LIN {X 0,Y 458.208,Z 900.819,A -85,B 0,C 180,E1 13122.077,E2 13122.077} C_VEL
LIN {X 0,Y 454.402,Z 922.56,A -85,B 0,C 180,E1 13121.642,E2 13121.642} C_VEL
LIN {X 0,Y 449.592,Z 944.659,A -85,B 0,C 180,E1 13121.087,E2 13121.087} C_VEL
LIN {X 0,Y 442.831,Z 970.318,A -85,B 0,C 180,E1 13120.289,E2 13120.289} C_VEL
LIN {X 0,Y 434.901,Z 994.961,A -85,B 0,C 180,E1 13119.322,E2 13119.322} C_VEL
LIN {X 0,Y 427.473,Z 1015.224,A -85,B 0,C 180,E1 13118.375,E2 13118.375} C_VEL
LIN {X 0,Y 419.408,Z 1034.951,A -85,B 0,C 180,E1 13117.289,E2 13117.289} C_VEL
LIN {X 0,Y 409.247,Z 1057.358,A -85,B 0,C 180,E1 13115.837,E2 13115.837} C_VEL
LIN {X 0,Y 397.642,Z 1080.077,A -85,B 0,C 180,E1 13114.053,E2 13114.053} C_VEL
LIN {X 0,Y 387.753,Z 1097.858,A -85,B 0,C 180,E1 13112.398,E2 13112.398} C_VEL
LIN {X 0,Y 377.989,Z 1114.238,A -85,B 0,C 180,E1 13110.628,E2 13110.628} C_VEL
LIN {X 0,Y 368.063,Z 1129.874,A -85,B 0,C 180,E1 13108.672,E2 13108.672} C_VEL
LIN {X 0,Y 355.822,Z 1148.166,A -85,B 0,C 180,E1 13105.975,E2 13105.975} C_VEL
LIN {X 0,Y 343.486,Z 1165.363,A -85,B 0,C 180,E1 13102.886,E2 13102.886} C_VEL
LIN {X 0,Y 333.685,Z 1178.527,A -85,B 0,C 180,E1 13100.078,E2 13100.078} C_VEL
LIN {X 0,Y 324.574,Z 1190.478,A -85,B 0,C 180,E1 13097.092,E2 13097.092} C_VEL
LIN {X 0,Y 315.879,Z 1201.713,A -85,B 0,C 180,E1 13093.803,E2 13093.803} C_VEL
LIN {X 0,Y 306.032,Z 1214.541,A -85,B 0,C 180,E1 13089.321,E2 13089.321} C_VEL
LIN {X 0,Y 297.777,Z 1225.367,A -85,B 0,C 180,E1 13084.561,E2 13084.561} C_VEL
LIN {X 0,Y 292.177,Z 1233.181,A -85,B 0,C 180,E1 13080.413,E2 13080.413} C_VEL
LIN {X 0,Y 287.782,Z 1239.822,A -85,B 0,C 180,E1 13076.172,E2 13076.172} C_VEL
LIN {X 0,Y 284.237,Z 1245.857,A -85,B 0,C 180,E1 13071.449,E2 13071.449} C_VEL
LIN {X 0,Y 281.638,Z 1251.335,A -85,B 0,C 180,E1 13065.819,E2 13065.819} C_VEL
LIN {X 0,Y 280.53,Z 1254.566,A -85,B 0,C 180,E1 13061.087,E2 13061.087} C_VEL
LIN {X 0,Y 280.133,Z 1256.541,A -85,B 0,C 180,E1 13056.755,E2 13056.755} C_VEL
LIN {X 0,Y 280.008,Z 1257.539,A -85,B 0,C 180,E1 13052.651,E2 13052.651} C_VEL
LIN {X 0,Y 279.986,Z 1257.679,A -85,B 0,C 180,E1 13048.558,E2 13048.558} C_VEL
LIN {X 0,Y 280.068,Z 1256.959,A -85,B 0,C 180,E1 13044.459,E2 13044.459} C_VEL
LIN {X 0,Y 280.331,Z 1255.374,A -85,B 0,C 180,E1 13040.34,E2 13040.34} C_VEL
LIN {X 0,Y 281.103,Z 1252.753,A -85,B 0,C 180,E1 13035.994,E2 13035.994} C_VEL
LIN {X 0,Y 282.595,Z 1249.134,A -85,B 0,C 180,E1 13031.636,E2 13031.636} C_VEL
LIN {X 0,Y 284.991,Z 1244.486,A -85,B 0,C 180,E1 13027.29,E2 13027.29} C_VEL
LIN {X 0,Y 288.66,Z 1238.479,A -85,B 0,C 180,E1 13022.783,E2 13022.783} C_VEL
LIN {X 0,Y 294.638,Z 1229.864,A -85,B 0,C 180,E1 13017.567,E2 13017.567} C_VEL
LIN {X 0,Y 302.104,Z 1219.641,A -85,B 0,C 180,E1 13012.714,E2 13012.714} C_VEL
LIN {X 0,Y 309.339,Z 1210.213,A -85,B 0,C 180,E1 13008.984,E2 13008.984} C_VEL
LIN {X 0,Y 317.621,Z 1199.529,A -85,B 0,C 180,E1 13005.403,E2 13005.403} C_VEL
LIN {X 0,Y 328.464,Z 1185.62,A -85,B 0,C 180,E1 13001.5,E2 13001.5} C_VEL
LIN {X 0,Y 340.404,Z 1169.657,A -85,B 0,C 180,E1 12997.873,E2 12997.873} C_VEL
LIN {X 0,Y 350.282,Z 1156.036,A -85,B 0,C 180,E1 12995.266,E2 12995.266} C_VEL
LIN {X 0,Y 359.989,Z 1142.109,A -85,B 0,C 180,E1 12992.976,E2 12992.976} C_VEL
LIN {X 0,Y 370.544,Z 1126.229,A -85,B 0,C 180,E1 12990.737,E2 12990.737} C_VEL
LIN {X 0,Y 383.441,Z 1105.562,A -85,B 0,C 180,E1 12988.284,E2 12988.284} C_VEL
LIN {X 0,Y 394.996,Z 1085.203,A -85,B 0,C 180,E1 12986.295,E2 12986.295} C_VEL
LIN {X 0,Y 404.338,Z 1067.469,A -85,B 0,C 180,E1 12984.822,E2 12984.822} C_VEL
LIN {X 0,Y 412.871,Z 1049.87,A -85,B 0,C 180,E1 12983.553,E2 12983.553} C_VEL
LIN {X 0,Y 416.305,Z 1042.588,A -85,B 0,C 180,E1 12983.075,E2 12983.075} C_VEL
LIN {X 0,Y 418.753,Z 1036.276,A -85,B 0,C 180,E1 12982.553,E2 12982.553} C_VEL
LIN {X 0,Y 423.276,Z 1019.851,A -85,B 0,C 180,E1 12980.83,E2 12980.83} C_VEL
LIN {X 0,Y 425.239,Z 1014.185,A -85,B 0,C 180,E1 12980.445,E2 12980.445} C_VEL
LIN {X 0,Y 433.639,Z 991.447,A -85,B 0,C 180,E1 12979.417,E2 12979.417} C_VEL
LIN {X 0,Y 441.922,Z 964.972,A -85,B 0,C 180,E1 12978.443,E2 12978.443} C_VEL
LIN {X 0,Y 447.766,Z 942.648,A -85,B 0,C 180,E1 12977.78,E2 12977.78} C_VEL
LIN {X 0,Y 452.432,Z 921.238,A -85,B 0,C 180,E1 12977.26,E2 12977.26} C_VEL
LIN {X 0,Y 456.431,Z 898.287,A -85,B 0,C 180,E1 12976.818,E2 12976.818} C_VEL
LIN {X 0,Y 460.408,Z 864.162,A -85,B 0,C 180,E1 12976.277,E2 12976.277} C_VEL
LIN {X 0,Y 479.796,Z 660.807,A -85,B 0,C 180,E1 12973.266,E2 12973.266} C_VEL
LIN {X 0,Y 476.185,Z 654.134,A -85,B 0,C 180,E1 12970.71,E2 12970.71} C_VEL
LIN {X 0,Y 473.814,Z 649.968,A -85,B 0,C 180,E1 12968.617,E2 12968.617} C_VEL
LIN {X 0,Y 471.686,Z 646,A -85,B 0,C 180,E1 12966.084,E2 12966.084} C_VEL
LIN {X 0,Y 469.89,Z 641.972,A -85,B 0,C 180,E1 12961.829,E2 12961.829} C_VEL
LIN {X 0,Y 469.82,Z 641.352,A -85,B 0,C 180,E1 12960.976,E2 12960.976} C_VEL
LIN {X 0,Y 469.873,Z 641.573,A -85,B 0,C 180,E1 12958.903,E2 12958.903} C_VEL
LIN {X 0,Y 471.37,Z 645.689,A -85,B 0,C 180,E1 12954.767,E2 12954.767} C_VEL
LIN {X 0,Y 472.117,Z 646.8,A -85,B 0,C 180,E1 12953.738,E2 12953.738} C_VEL
LIN {X 0,Y 474.753,Z 651.624,A -85,B 0,C 180,E1 12950.912,E2 12950.912} C_VEL
LIN {X 0,Y 477.243,Z 656.203,A -85,B 0,C 180,E1 12948.886,E2 12948.886} C_VEL
LIN {X 0,Y 479.059,Z 659.618,A -85,B 0,C 180,E1 12947.616,E2 12947.616} C_VEL
LIN {X 0,Y 479.91,Z 661.708,A -85,B 0,C 180,E1 12947.034,E2 12947.034} C_VEL
LIN {X 0,Y 459.294,Z 878.88,A -85,B 0,C 180,E1 12943.812,E2 12943.812} C_VEL
LIN {X 0,Y 455.731,Z 908,A -85,B 0,C 180,E1 12943.338,E2 12943.338} C_VEL
LIN {X 0,Y 451.723,Z 930.654,A -85,B 0,C 180,E1 12942.918,E2 12942.918} C_VEL
LIN {X 0,Y 446.837,Z 952.503,A -85,B 0,C 180,E1 12942.435,E2 12942.435} C_VEL
LIN {X 0,Y 440.026,Z 977.894,A -85,B 0,C 180,E1 12941.725,E2 12941.725} C_VEL
LIN {X 0,Y 431.647,Z 1003.54,A -85,B 0,C 180,E1 12940.813,E2 12940.813} C_VEL
LIN {X 0,Y 423.793,Z 1024.563,A -85,B 0,C 180,E1 12939.899,E2 12939.899} C_VEL
LIN {X 0,Y 415.815,Z 1043.731,A -85,B 0,C 180,E1 12938.917,E2 12938.917} C_VEL
LIN {X 0,Y 406.864,Z 1063.298,A -85,B 0,C 180,E1 12937.736,E2 12937.736} C_VEL
LIN {X 0,Y 395.004,Z 1086.874,A -85,B 0,C 180,E1 12936.046,E2 12936.046} C_VEL
LIN {X 0,Y 382.76,Z 1108.625,A -85,B 0,C 180,E1 12934.135,E2 12934.135} C_VEL
LIN {X 0,Y 372.487,Z 1125.659,A -85,B 0,C 180,E1 12932.364,E2 12932.364} C_VEL
LIN {X 0,Y 361.948,Z 1142.122,A -85,B 0,C 180,E1 12930.364,E2 12930.364} C_VEL
LIN {X 0,Y 349.824,Z 1160.077,A -85,B 0,C 180,E1 12927.793,E2 12927.793} C_VEL
LIN {X 0,Y 336.403,Z 1178.724,A -85,B 0,C 180,E1 12924.538,E2 12924.538} C_VEL
LIN {X 0,Y 326.264,Z 1192.331,A -85,B 0,C 180,E1 12921.688,E2 12921.688} C_VEL
LIN {X 0,Y 316.923,Z 1204.607,A -85,B 0,C 180,E1 12918.676,E2 12918.676} C_VEL
LIN {X 0,Y 307.429,Z 1216.966,A -85,B 0,C 180,E1 12915.107,E2 12915.107} C_VEL
LIN {X 0,Y 296.996,Z 1230.755,A -85,B 0,C 180,E1 12910.279,E2 12910.279} C_VEL
LIN {X 0,Y 289.063,Z 1241.475,A -85,B 0,C 180,E1 12905.621,E2 12905.621} C_VEL
LIN {X 0,Y 283.333,Z 1249.819,A -85,B 0,C 180,E1 12901.258,E2 12901.258} C_VEL
LIN {X 0,Y 278.777,Z 1257.144,A -85,B 0,C 180,E1 12896.646,E2 12896.646} C_VEL
LIN {X 0,Y 274.966,Z 1264.468,A -85,B 0,C 180,E1 12890.886,E2 12890.886} C_VEL
LIN {X 0,Y 273.019,Z 1269.339,A -85,B 0,C 180,E1 12885.734,E2 12885.734} C_VEL
LIN {X 0,Y 272.243,Z 1272.504,A -85,B 0,C 180,E1 12881.234,E2 12881.234} C_VEL
LIN {X 0,Y 272.013,Z 1274.548,A -85,B 0,C 180,E1 12876.977,E2 12876.977} C_VEL
LIN {X 0,Y 271.992,Z 1275.618,A -85,B 0,C 180,E1 12872.96,E2 12872.96} C_VEL
LIN {X 0,Y 271.98,Z 1275.809,A -85,B 0,C 180,E1 12868.746,E2 12868.746} C_VEL
LIN {X 0,Y 271.99,Z 1275.049,A -85,B 0,C 180,E1 12864.525,E2 12864.525} C_VEL
LIN {X 0,Y 272.086,Z 1273.337,A -85,B 0,C 180,E1 12860.278,E2 12860.278} C_VEL
LIN {X 0,Y 272.693,Z 1270.509,A -85,B 0,C 180,E1 12855.789,E2 12855.789} C_VEL
LIN {X 0,Y 274.01,Z 1266.621,A -85,B 0,C 180,E1 12851.28,E2 12851.28} C_VEL
LIN {X 0,Y 276.262,Z 1261.652,A -85,B 0,C 180,E1 12846.776,E2 12846.776} C_VEL
LIN {X 0,Y 279.474,Z 1255.891,A -85,B 0,C 180,E1 12842.526,E2 12842.526} C_VEL
LIN {X 0,Y 284.029,Z 1248.723,A -85,B 0,C 180,E1 12838.139,E2 12838.139} C_VEL
LIN {X 0,Y 291.432,Z 1238.275,A -85,B 0,C 180,E1 12832.868,E2 12832.868} C_VEL
LIN {X 0,Y 300.371,Z 1226.138,A -85,B 0,C 180,E1 12828.017,E2 12828.017} C_VEL
LIN {X 0,Y 308.826,Z 1215.076,A -85,B 0,C 180,E1 12824.329,E2 12824.329} C_VEL
LIN {X 0,Y 318.374,Z 1202.649,A -85,B 0,C 180,E1 12820.826,E2 12820.826} C_VEL
LIN {X 0,Y 330.9,Z 1186.15,A -85,B 0,C 180,E1 12816.965,E2 12816.965} C_VEL
LIN {X 0,Y 342.902,Z 1169.616,A -85,B 0,C 180,E1 12813.812,E2 12813.812} C_VEL
LIN {X 0,Y 353.575,Z 1154.399,A -85,B 0,C 180,E1 12811.366,E2 12811.366} C_VEL
LIN {X 0,Y 364.164,Z 1138.584,A -85,B 0,C 180,E1 12809.196,E2 12809.196} C_VEL
LIN {X 0,Y 377.019,Z 1118.286,A -85,B 0,C 180,E1 12806.842,E2 12806.842} C_VEL
LIN {X 0,Y 389.335,Z 1096.889,A -85,B 0,C 180,E1 12804.812,E2 12804.812} C_VEL
LIN {X 0,Y 399.1,Z 1078.591,A -85,B 0,C 180,E1 12803.34,E2 12803.34} C_VEL
LIN {X 0,Y 408.668,Z 1059.163,A -85,B 0,C 180,E1 12802.008,E2 12802.008} C_VEL
LIN {X 0,Y 418.509,Z 1037.249,A -85,B 0,C 180,E1 12800.74,E2 12800.74} C_VEL
LIN {X 0,Y 428.549,Z 1011.748,A -85,B 0,C 180,E1 12799.533,E2 12799.533} C_VEL
LIN {X 0,Y 435.907,Z 990.374,A -85,B 0,C 180,E1 12798.705,E2 12798.705} C_VEL
LIN {X 0,Y 441.98,Z 970.274,A -85,B 0,C 180,E1 12798.055,E2 12798.055} C_VEL
LIN {X 0,Y 447.636,Z 948.487,A -85,B 0,C 180,E1 12797.476,E2 12797.476} C_VEL
LIN {X 0,Y 453.046,Z 923.261,A -85,B 0,C 180,E1 12796.943,E2 12796.943} C_VEL
LIN {X 0,Y 457.356,Z 894.787,A -85,B 0,C 180,E1 12796.445,E2 12796.445} C_VEL
LIN {X 0,Y 464.969,Z 816.08,A -85,B 0,C 180,E1 12795.257,E2 12795.257} C_VEL
LIN {X 0,Y 479.707,Z 661.387,A -85,B 0,C 180,E1 12792.948,E2 12792.948} C_VEL
LIN {X 0,Y 477.878,Z 657.566,A -85,B 0,C 180,E1 12791.71,E2 12791.71} C_VEL
LIN {X 0,Y 475.155,Z 652.651,A -85,B 0,C 180,E1 12789.631,E2 12789.631} C_VEL
LIN {X 0,Y 473.644,Z 649.962,A -85,B 0,C 180,E1 12788.253,E2 12788.253} C_VEL
LIN {X 0,Y 471.486,Z 645.953,A -85,B 0,C 180,E1 12785.72,E2 12785.72} C_VEL
LIN {X 0,Y 469.719,Z 642.322,A -85,B 0,C 180,E1 12781.952,E2 12781.952} C_VEL
LIN {X 0,Y 469.602,Z 641.325,A -85,B 0,C 180,E1 12780.976,E2 12780.976} C_VEL
LIN {X 0,Y 469.642,Z 641.564,A -85,B 0,C 180,E1 12778.17,E2 12778.17} C_VEL
LIN {X 0,Y 471.383,Z 645.828,A -85,B 0,C 180,E1 12773.912,E2 12773.912} C_VEL
LIN {X 0,Y 472.055,Z 647.057,A -85,B 0,C 180,E1 12773.004,E2 12773.004} C_VEL
LIN {X 0,Y 474.46,Z 651.334,A -85,B 0,C 180,E1 12770.478,E2 12770.478} C_VEL
LIN {X 0,Y 477.27,Z 656.469,A -85,B 0,C 180,E1 12768.213,E2 12768.213} C_VEL
LIN {X 0,Y 479.605,Z 660.806,A -85,B 0,C 180,E1 12766.635,E2 12766.635} C_VEL
LIN {X 0,Y 458.7,Z 879.164,A -85,B 0,C 180,E1 12763.397,E2 12763.397} C_VEL
LIN {X 0,Y 455.655,Z 902.058,A -85,B 0,C 180,E1 12763.018,E2 12763.018} C_VEL
LIN {X 0,Y 451.751,Z 923.802,A -85,B 0,C 180,E1 12762.585,E2 12762.585} C_VEL
LIN {X 0,Y 446.411,Z 947.667,A -85,B 0,C 180,E1 12761.986,E2 12761.986} C_VEL
LIN {X 0,Y 438.836,Z 974.812,A -85,B 0,C 180,E1 12761.122,E2 12761.122} C_VEL
LIN {X 0,Y 431.717,Z 996.356,A -85,B 0,C 180,E1 12760.275,E2 12760.275} C_VEL
LIN {X 0,Y 424.163,Z 1016.494,A -85,B 0,C 180,E1 12759.34,E2 12759.34} C_VEL
LIN {X 0,Y 416.019,Z 1035.968,A -85,B 0,C 180,E1 12758.276,E2 12758.276} C_VEL
LIN {X 0,Y 404.868,Z 1059.921,A -85,B 0,C 180,E1 12756.725,E2 12756.725} C_VEL
LIN {X 0,Y 393.273,Z 1081.892,A -85,B 0,C 180,E1 12754.989,E2 12754.989} C_VEL
LIN {X 0,Y 383.503,Z 1099.004,A -85,B 0,C 180,E1 12753.395,E2 12753.395} C_VEL
LIN {X 0,Y 373.675,Z 1115.061,A -85,B 0,C 180,E1 12751.663,E2 12751.663} C_VEL
LIN {X 0,Y 362.847,Z 1131.649,A -85,B 0,C 180,E1 12749.581,E2 12749.581} C_VEL
LIN {X 0,Y 349.383,Z 1151.011,A -85,B 0,C 180,E1 12746.667,E2 12746.667} C_VEL
LIN {X 0,Y 337.953,Z 1166.396,A -85,B 0,C 180,E1 12743.855,E2 12743.855} C_VEL
LIN {X 0,Y 327.862,Z 1179.49,A -85,B 0,C 180,E1 12741.032,E2 12741.032} C_VEL
LIN {X 0,Y 318.054,Z 1191.887,A -85,B 0,C 180,E1 12737.88,E2 12737.88} C_VEL
LIN {X 0,Y 307.077,Z 1205.615,A -85,B 0,C 180,E1 12733.708,E2 12733.708} C_VEL
LIN {X 0,Y 297.378,Z 1217.505,A -85,B 0,C 180,E1 12729.193,E2 12729.193} C_VEL
LIN {X 0,Y 290.336,Z 1226.43,A -85,B 0,C 180,E1 12725.095,E2 12725.095} C_VEL
LIN {X 0,Y 284.549,Z 1234.133,A -85,B 0,C 180,E1 12720.853,E2 12720.853} C_VEL
LIN {X 0,Y 279.442,Z 1241.562,A -85,B 0,C 180,E1 12715.871,E2 12715.871} C_VEL
LIN {X 0,Y 275.381,Z 1248.326,A -85,B 0,C 180,E1 12709.945,E2 12709.945} C_VEL
LIN {X 0,Y 273.434,Z 1252.438,A -85,B 0,C 180,E1 12705.117,E2 12705.117} C_VEL
LIN {X 0,Y 272.515,Z 1255.049,A -85,B 0,C 180,E1 12700.989,E2 12700.989} C_VEL
LIN {X 0,Y 272.138,Z 1256.869,A -85,B 0,C 180,E1 12696.742,E2 12696.742} C_VEL
LIN {X 0,Y 272.013,Z 1257.802,A -85,B 0,C 180,E1 12692.729,E2 12692.729} C_VEL
LIN {X 0,Y 271.983,Z 1257.964,A -85,B 0,C 180,E1 12688.727,E2 12688.727} C_VEL
LIN {X 0,Y 272.072,Z 1257.287,A -85,B 0,C 180,E1 12684.508,E2 12684.508} C_VEL
LIN {X 0,Y 272.363,Z 1255.639,A -85,B 0,C 180,E1 12680.055,E2 12680.055} C_VEL
LIN {X 0,Y 273.215,Z 1253.019,A -85,B 0,C 180,E1 12675.581,E2 12675.581} C_VEL
LIN {X 0,Y 274.835,Z 1249.378,A -85,B 0,C 180,E1 12671.071,E2 12671.071} C_VEL
LIN {X 0,Y 277.395,Z 1244.756,A -85,B 0,C 180,E1 12666.632,E2 12666.632} C_VEL
LIN {X 0,Y 281.107,Z 1239.043,A -85,B 0,C 180,E1 12662.219,E2 12662.219} C_VEL
LIN {X 0,Y 287.107,Z 1230.825,A -85,B 0,C 180,E1 12657.069,E2 12657.069} C_VEL
LIN {X 0,Y 295.163,Z 1220.361,A -85,B 0,C 180,E1 12651.927,E2 12651.927} C_VEL
LIN {X 0,Y 303.082,Z 1210.485,A -85,B 0,C 180,E1 12647.947,E2 12647.947} C_VEL
LIN {X 0,Y 311.727,Z 1199.801,A -85,B 0,C 180,E1 12644.325,E2 12644.325} C_VEL
LIN {X 0,Y 323.002,Z 1185.891,A -85,B 0,C 180,E1 12640.393,E2 12640.393} C_VEL
LIN {X 0,Y 334.962,Z 1170.462,A -85,B 0,C 180,E1 12636.861,E2 12636.861} C_VEL
LIN {X 0,Y 345.562,Z 1156.305,A -85,B 0,C 180,E1 12634.144,E2 12634.144} C_VEL
LIN {X 0,Y 356.201,Z 1141.464,A -85,B 0,C 180,E1 12631.72,E2 12631.72} C_VEL
LIN {X 0,Y 368.389,Z 1123.555,A -85,B 0,C 180,E1 12629.246,E2 12629.246} C_VEL
LIN {X 0,Y 381.61,Z 1102.427,A -85,B 0,C 180,E1 12626.844,E2 12626.844} C_VEL
LIN {X 0,Y 392.067,Z 1084.328,A -85,B 0,C 180,E1 12625.12,E2 12625.12} C_VEL
LIN {X 0,Y 401.727,Z 1066.276,A -85,B 0,C 180,E1 12623.651,E2 12623.651} C_VEL
LIN {X 0,Y 410.852,Z 1047.707,A -85,B 0,C 180,E1 12622.352,E2 12622.352} C_VEL
LIN {X 0,Y 421.721,Z 1023.115,A -85,B 0,C 180,E1 12620.898,E2 12620.898} C_VEL
LIN {X 0,Y 425.239,Z 1014.185,A -85,B 0,C 180,E1 12620.445,E2 12620.445} C_VEL
LIN {X 0,Y 427.575,Z 1007.549,A -85,B 0,C 180,E1 12619.999,E2 12619.999} C_VEL
LIN {X 0,Y 431.528,Z 991.264,A -85,B 0,C 180,E1 12618.513,E2 12618.513} C_VEL
LIN {X 0,Y 433.488,Z 984.381,A -85,B 0,C 180,E1 12618.119,E2 12618.119} C_VEL
LIN {X 0,Y 440.062,Z 963.018,A -85,B 0,C 180,E1 12617.378,E2 12617.378} C_VEL
LIN {X 0,Y 445.664,Z 941.713,A -85,B 0,C 180,E1 12616.764,E2 12616.764} C_VEL
LIN {X 0,Y 450.436,Z 919.913,A -85,B 0,C 180,E1 12616.252,E2 12616.252} C_VEL
LIN {X 0,Y 455.094,Z 892.816,A -85,B 0,C 180,E1 12615.752,E2 12615.752} C_VEL
LIN {X 0,Y 459.703,Z 848.917,A -85,B 0,C 180,E1 12615.086,E2 12615.086} C_VEL
LIN {X 0,Y 477.447,Z 666.619,A -85,B 0,C 180,E1 12612.402,E2 12612.402} C_VEL
LIN {X 0,Y 474.383,Z 661,A -85,B 0,C 180,E1 12610.076,E2 12610.076} C_VEL
LIN {X 0,Y 472.589,Z 657.681,A -85,B 0,C 180,E1 12608.395,E2 12608.395} C_VEL
LIN {X 0,Y 470.622,Z 653.883,A -85,B 0,C 180,E1 12605.976,E2 12605.976} C_VEL
LIN {X 0,Y 468.896,Z 649.851,A -85,B 0,C 180,E1 12601.711,E2 12601.711} C_VEL
LIN {X 0,Y 468.833,Z 649.296,A -85,B 0,C 180,E1 12600.855,E2 12600.855} C_VEL
LIN {X 0,Y 468.888,Z 649.598,A -85,B 0,C 180,E1 12598.9,E2 12598.9} C_VEL
LIN {X 0,Y 470.395,Z 653.667,A -85,B 0,C 180,E1 12594.756,E2 12594.756} C_VEL
LIN {X 0,Y 471.081,Z 654.828,A -85,B 0,C 180,E1 12593.786,E2 12593.786} C_VEL
LIN {X 0,Y 473.565,Z 659.444,A -85,B 0,C 180,E1 12591.072,E2 12591.072} C_VEL
LIN {X 0,Y 476.005,Z 664.046,A -85,B 0,C 180,E1 12589.041,E2 12589.041} C_VEL
LIN {X 0,Y 477.6,Z 667.148,A -85,B 0,C 180,E1 12587.894,E2 12587.894} C_VEL
LIN {X 0,Y 456.821,Z 881.666,A -85,B 0,C 180,E1 12584.736,E2 12584.736} C_VEL
LIN {X 0,Y 453.331,Z 908.729,A -85,B 0,C 180,E1 12584.296,E2 12584.296} C_VEL
LIN {X 0,Y 449.294,Z 931.036,A -85,B 0,C 180,E1 12583.887,E2 12583.887} C_VEL
LIN {X 0,Y 444.21,Z 953.307,A -85,B 0,C 180,E1 12583.401,E2 12583.401} C_VEL
LIN {X 0,Y 436.833,Z 980.014,A -85,B 0,C 180,E1 12582.658,E2 12582.658} C_VEL
LIN {X 0,Y 428.5,Z 1004.768,A -85,B 0,C 180,E1 12581.779,E2 12581.779} C_VEL
LIN {X 0,Y 421.059,Z 1024.302,A -85,B 0,C 180,E1 12580.941,E2 12580.941} C_VEL
LIN {X 0,Y 412.941,Z 1043.468,A -85,B 0,C 180,E1 12579.977,E2 12579.977} C_VEL
LIN {X 0,Y 403.697,Z 1063.286,A -85,B 0,C 180,E1 12578.8,E2 12578.8} C_VEL
LIN {X 0,Y 391.722,Z 1086.607,A -85,B 0,C 180,E1 12577.151,E2 12577.151} C_VEL
LIN {X 0,Y 379.266,Z 1108.269,A -85,B 0,C 180,E1 12575.271,E2 12575.271} C_VEL
LIN {X 0,Y 368.342,Z 1125.951,A -85,B 0,C 180,E1 12573.447,E2 12573.447} C_VEL
LIN {X 0,Y 357.473,Z 1142.472,A -85,B 0,C 180,E1 12571.446,E2 12571.446} C_VEL
LIN {X 0,Y 344.129,Z 1161.658,A -85,B 0,C 180,E1 12568.684,E2 12568.684} C_VEL
LIN {X 0,Y 330.986,Z 1179.233,A -85,B 0,C 180,E1 12565.569,E2 12565.569} C_VEL
LIN {X 0,Y 320.542,Z 1192.769,A -85,B 0,C 180,E1 12562.706,E2 12562.706} C_VEL
LIN {X 0,Y 310.381,Z 1205.626,A -85,B 0,C 180,E1 12559.497,E2 12559.497} C_VEL
LIN {X 0,Y 298.908,Z 1220.065,A -85,B 0,C 180,E1 12555.176,E2 12555.176} C_VEL
LIN {X 0,Y 288.683,Z 1232.832,A -85,B 0,C 180,E1 12550.377,E2 12550.377} C_VEL
LIN {X 0,Y 281.829,Z 1241.758,A -85,B 0,C 180,E1 12546.343,E2 12546.343} C_VEL
LIN {X 0,Y 275.935,Z 1249.908,A -85,B 0,C 180,E1 12541.95,E2 12541.95} C_VEL
LIN {X 0,Y 270.788,Z 1257.81,A -85,B 0,C 180,E1 12536.784,E2 12536.784} C_VEL
LIN {X 0,Y 266.909,Z 1264.843,A -85,B 0,C 180,E1 12530.857,E2 12530.857} C_VEL
LIN {X 0,Y 265.074,Z 1269.238,A -85,B 0,C 180,E1 12525.993,E2 12525.993} C_VEL
LIN {X 0,Y 264.272,Z 1272.283,A -85,B 0,C 180,E1 12521.493,E2 12521.493} C_VEL
LIN {X 0,Y 264.019,Z 1274.301,A -85,B 0,C 180,E1 12517.138,E2 12517.138} C_VEL
LIN {X 0,Y 263.995,Z 1275.355,A -85,B 0,C 180,E1 12513.049,E2 12513.049} C_VEL
LIN {X 0,Y 263.986,Z 1275.546,A -85,B 0,C 180,E1 12508.708,E2 12508.708} C_VEL
LIN {X 0,Y 263.994,Z 1274.785,A -85,B 0,C 180,E1 12504.359,E2 12504.359} C_VEL
LIN {X 0,Y 264.107,Z 1273.071,A -85,B 0,C 180,E1 12499.981,E2 12499.981} C_VEL
LIN {X 0,Y 264.777,Z 1270.24,A -85,B 0,C 180,E1 12495.355,E2 12495.355} C_VEL
LIN {X 0,Y 266.215,Z 1266.349,A -85,B 0,C 180,E1 12490.711,E2 12490.711} C_VEL
LIN {X 0,Y 268.649,Z 1261.379,A -85,B 0,C 180,E1 12486.078,E2 12486.078} C_VEL
LIN {X 0,Y 272.078,Z 1255.615,A -85,B 0,C 180,E1 12481.714,E2 12481.714} C_VEL
LIN {X 0,Y 276.916,Z 1248.445,A -85,B 0,C 180,E1 12477.219,E2 12477.219} C_VEL
LIN {X 0,Y 284.745,Z 1237.996,A -85,B 0,C 180,E1 12471.842,E2 12471.842} C_VEL
LIN {X 0,Y 294.143,Z 1225.859,A -85,B 0,C 180,E1 12466.916,E2 12466.916} C_VEL
LIN {X 0,Y 302.986,Z 1214.797,A -85,B 0,C 180,E1 12463.186,E2 12463.186} C_VEL
LIN {X 0,Y 312.522,Z 1202.855,A -85,B 0,C 180,E1 12459.783,E2 12459.783} C_VEL
LIN {X 0,Y 325.254,Z 1186.74,A -85,B 0,C 180,E1 12455.957,E2 12455.957} C_VEL
LIN {X 0,Y 337.665,Z 1170.196,A -85,B 0,C 180,E1 12452.776,E2 12452.776} C_VEL
LIN {X 0,Y 348.727,Z 1154.907,A -85,B 0,C 180,E1 12450.307,E2 12450.307} C_VEL
LIN {X 0,Y 359.467,Z 1139.333,A -85,B 0,C 180,E1 12448.166,E2 12448.166} C_VEL
LIN {X 0,Y 370.356,Z 1122.62,A -85,B 0,C 180,E1 12446.202,E2 12446.202} C_VEL
LIN {X 0,Y 384.054,Z 1099.985,A -85,B 0,C 180,E1 12443.984,E2 12443.984} C_VEL
LIN {X 0,Y 395.093,Z 1079.872,A -85,B 0,C 180,E1 12442.358,E2 12442.358} C_VEL
LIN {X 0,Y 404.869,Z 1060.524,A -85,B 0,C 180,E1 12441.035,E2 12441.035} C_VEL
LIN {X 0,Y 414.021,Z 1040.69,A -85,B 0,C 180,E1 12439.884,E2 12439.884} C_VEL
LIN {X 0,Y 424.257,Z 1016.016,A -85,B 0,C 180,E1 12438.689,E2 12438.689} C_VEL
LIN {X 0,Y 432.956,Z 991.392,A -85,B 0,C 180,E1 12437.733,E2 12437.733} C_VEL
LIN {X 0,Y 439.337,Z 970.713,A -85,B 0,C 180,E1 12437.073,E2 12437.073} C_VEL
LIN {X 0,Y 444.987,Z 949.409,A -85,B 0,C 180,E1 12436.514,E2 12436.514} C_VEL
LIN {X 0,Y 449.988,Z 926.777,A -85,B 0,C 180,E1 12436.037,E2 12436.037} C_VEL
LIN {X 0,Y 454.779,Z 897.617,A -85,B 0,C 180,E1 12435.522,E2 12435.522} C_VEL
LIN {X 0,Y 459.902,Z 847.321,A -85,B 0,C 180,E1 12434.762,E2 12434.762} C_VEL
LIN {X 0,Y 477.403,Z 667.033,A -85,B 0,C 180,E1 12432.107,E2 12432.107} C_VEL
LIN {X 0,Y 474.528,Z 661.442,A -85,B 0,C 180,E1 12429.95,E2 12429.95} C_VEL
LIN {X 0,Y 472.415,Z 657.674,A -85,B 0,C 180,E1 12428.03,E2 12428.03} C_VEL
LIN {X 0,Y 470.42,Z 653.834,A -85,B 0,C 180,E1 12425.611,E2 12425.611} C_VEL
LIN {X 0,Y 468.698,Z 650.05,A -85,B 0,C 180,E1 12421.711,E2 12421.711} C_VEL
LIN {X 0,Y 468.606,Z 649.27,A -85,B 0,C 180,E1 12420.856,E2 12420.856} C_VEL
LIN {X 0,Y 468.648,Z 649.446,A -85,B 0,C 180,E1 12418.288,E2 12418.288} C_VEL
LIN {X 0,Y 470.32,Z 653.709,A -85,B 0,C 180,E1 12414.02,E2 12414.02} C_VEL
LIN {X 0,Y 471.11,Z 655.294,A -85,B 0,C 180,E1 12412.929,E2 12412.929} C_VEL
LIN {X 0,Y 473.272,Z 659.16,A -85,B 0,C 180,E1 12410.637,E2 12410.637} C_VEL
LIN {X 0,Y 475.949,Z 664.164,A -85,B 0,C 180,E1 12408.426,E2 12408.426} C_VEL
LIN {X 0,Y 477.259,Z 666.712,A -85,B 0,C 180,E1 12407.488,E2 12407.488} C_VEL
LIN {X 0,Y 456.221,Z 881.637,A -85,B 0,C 180,E1 12404.326,E2 12404.326} C_VEL
LIN {X 0,Y 453.147,Z 903.794,A -85,B 0,C 180,E1 12403.96,E2 12403.96} C_VEL
LIN {X 0,Y 448.892,Z 926.703,A -85,B 0,C 180,E1 12403.502,E2 12403.502} C_VEL
LIN {X 0,Y 442.081,Z 955.209,A -85,B 0,C 180,E1 12402.765,E2 12402.765} C_VEL
LIN {X 0,Y 435.6,Z 977.25,A -85,B 0,C 180,E1 12402.044,E2 12402.044} C_VEL
LIN {X 0,Y 428.653,Z 997.752,A -85,B 0,C 180,E1 12401.242,E2 12401.242} C_VEL
LIN {X 0,Y 420.899,Z 1017.956,A -85,B 0,C 180,E1 12400.311,E2 12400.311} C_VEL
LIN {X 0,Y 411.308,Z 1040.285,A -85,B 0,C 180,E1 12399.084,E2 12399.084} C_VEL
LIN {X 0,Y 399.507,Z 1064.363,A -85,B 0,C 180,E1 12397.485,E2 12397.485} C_VEL
LIN {X 0,Y 389.136,Z 1083.487,A -85,B 0,C 180,E1 12395.964,E2 12395.964} C_VEL
LIN {X 0,Y 378.843,Z 1101.022,A -85,B 0,C 180,E1 12394.328,E2 12394.328} C_VEL
LIN {X 0,Y 367.209,Z 1119.444,A -85,B 0,C 180,E1 12392.309,E2 12392.309} C_VEL
LIN {X 0,Y 353.371,Z 1139.589,A -85,B 0,C 180,E1 12389.637,E2 12389.637} C_VEL
LIN {X 0,Y 342.352,Z 1154.615,A -85,B 0,C 180,E1 12387.242,E2 12387.242} C_VEL
LIN {X 0,Y 331.925,Z 1168.187,A -85,B 0,C 180,E1 12384.704,E2 12384.704} C_VEL
LIN {X 0,Y 321.58,Z 1181.142,A -85,B 0,C 180,E1 12381.856,E2 12381.856} C_VEL
LIN {X 0,Y 310.005,Z 1195.277,A -85,B 0,C 180,E1 12378.148,E2 12378.148} C_VEL
LIN {X 0,Y 298.311,Z 1209.064,A -85,B 0,C 180,E1 12373.653,E2 12373.653} C_VEL
LIN {X 0,Y 290.028,Z 1218.88,A -85,B 0,C 180,E1 12369.753,E2 12369.753} C_VEL
LIN {X 0,Y 282.826,Z 1227.611,A -85,B 0,C 180,E1 12365.597,E2 12365.597} C_VEL
LIN {X 0,Y 276.179,Z 1236.122,A -85,B 0,C 180,E1 12360.683,E2 12360.683} C_VEL
LIN {X 0,Y 270.548,Z 1243.945,A -85,B 0,C 180,E1 12354.906,E2 12354.906} C_VEL
LIN {X 0,Y 267.329,Z 1249.192,A -85,B 0,C 180,E1 12349.888,E2 12349.888} C_VEL
LIN {X 0,Y 265.481,Z 1252.915,A -85,B 0,C 180,E1 12345.275,E2 12345.275} C_VEL
LIN {X 0,Y 264.54,Z 1255.423,A -85,B 0,C 180,E1 12341.104,E2 12341.104} C_VEL
LIN {X 0,Y 264.143,Z 1257.198,A -85,B 0,C 180,E1 12336.729,E2 12336.729} C_VEL
LIN {X 0,Y 264.016,Z 1258.086,A -85,B 0,C 180,E1 12332.595,E2 12332.595} C_VEL
LIN {X 0,Y 263.997,Z 1258.204,A -85,B 0,C 180,E1 12328.471,E2 12328.471} C_VEL
LIN {X 0,Y 264.084,Z 1257.55,A -85,B 0,C 180,E1 12324.341,E2 12324.341} C_VEL
LIN {X 0,Y 264.4,Z 1255.904,A -85,B 0,C 180,E1 12319.752,E2 12319.752} C_VEL
LIN {X 0,Y 265.338,Z 1253.286,A -85,B 0,C 180,E1 12315.143,E2 12315.143} C_VEL
LIN {X 0,Y 267.074,Z 1249.671,A -85,B 0,C 180,E1 12310.527,E2 12310.527} C_VEL
LIN {X 0,Y 269.834,Z 1245.027,A -85,B 0,C 180,E1 12305.936,E2 12305.936} C_VEL
LIN {X 0,Y 273.794,Z 1239.314,A -85,B 0,C 180,E1 12301.409,E2 12301.409} C_VEL
LIN {X 0,Y 280.129,Z 1231.119,A -85,B 0,C 180,E1 12296.154,E2 12296.154} C_VEL
LIN {X 0,Y 288.692,Z 1220.574,A -85,B 0,C 180,E1 12290.881,E2 12290.881} C_VEL
LIN {X 0,Y 296.924,Z 1210.758,A -85,B 0,C 180,E1 12286.865,E2 12286.865} C_VEL
LIN {X 0,Y 305.953,Z 1200.073,A -85,B 0,C 180,E1 12283.206,E2 12283.206} C_VEL
LIN {X 0,Y 317.666,Z 1186.161,A -85,B 0,C 180,E1 12279.248,E2 12279.248} C_VEL
LIN {X 0,Y 330.043,Z 1170.732,A -85,B 0,C 180,E1 12275.707,E2 12275.707} C_VEL
LIN {X 0,Y 340.979,Z 1156.575,A -85,B 0,C 180,E1 12272.991,E2 12272.991} C_VEL
LIN {X 0,Y 351.986,Z 1141.65,A -85,B 0,C 180,E1 12270.563,E2 12270.563} C_VEL
LIN {X 0,Y 364.478,Z 1123.761,A -85,B 0,C 180,E1 12268.108,E2 12268.108} C_VEL
LIN {X 0,Y 377.613,Z 1103.294,A -85,B 0,C 180,E1 12265.795,E2 12265.795} C_VEL
LIN {X 0,Y 388.29,Z 1085.253,A -85,B 0,C 180,E1 12264.085,E2 12264.085} C_VEL
LIN {X 0,Y 398.139,Z 1067.267,A -85,B 0,C 180,E1 12262.631,E2 12262.631} C_VEL
LIN {X 0,Y 407.044,Z 1049.578,A -85,B 0,C 180,E1 12261.4,E2 12261.4} C_VEL
LIN {X 0,Y 416.5,Z 1028.913,A -85,B 0,C 180,E1 12260.161,E2 12260.161} C_VEL
LIN {X 0,Y 426.951,Z 1002.939,A -85,B 0,C 180,E1 12258.881,E2 12258.881} C_VEL
LIN {X 0,Y 433.488,Z 984.381,A -85,B 0,C 180,E1 12258.119,E2 12258.119} C_VEL
LIN {X 0,Y 435.46,Z 977.419,A -85,B 0,C 180,E1 12257.744,E2 12257.744} C_VEL
LIN {X 0,Y 439.077,Z 959.392,A -85,B 0,C 180,E1 12256.354,E2 12256.354} C_VEL
LIN {X 0,Y 440.585,Z 953.296,A -85,B 0,C 180,E1 12256.074,E2 12256.074} C_VEL
LIN {X 0,Y 447.07,Z 925.986,A -85,B 0,C 180,E1 12255.392,E2 12255.392} C_VEL
LIN {X 0,Y 451.261,Z 903.636,A -85,B 0,C 180,E1 12254.957,E2 12254.957} C_VEL
LIN {X 0,Y 454.386,Z 881.336,A -85,B 0,C 180,E1 12254.596,E2 12254.596} C_VEL
LIN {X 0,Y 475.219,Z 672.666,A -85,B 0,C 180,E1 12251.553,E2 12251.553} C_VEL
LIN {X 0,Y 472.842,Z 668.2,A -85,B 0,C 180,E1 12249.617,E2 12249.617} C_VEL
LIN {X 0,Y 471.371,Z 665.393,A -85,B 0,C 180,E1 12248.171,E2 12248.171} C_VEL
LIN {X 0,Y 469.56,Z 661.765,A -85,B 0,C 180,E1 12245.867,E2 12245.867} C_VEL
LIN {X 0,Y 467.903,Z 657.731,A -85,B 0,C 180,E1 12241.592,E2 12241.592} C_VEL
LIN {X 0,Y 467.858,Z 657.236,A -85,B 0,C 180,E1 12240.857,E2 12240.857} C_VEL
LIN {X 0,Y 467.899,Z 657.478,A -85,B 0,C 180,E1 12239.02,E2 12239.02} C_VEL
LIN {X 0,Y 469.337,Z 661.547,A -85,B 0,C 180,E1 12234.866,E2 12234.866} C_VEL
LIN {X 0,Y 470.004,Z 662.741,A -85,B 0,C 180,E1 12233.894,E2 12233.894} C_VEL
LIN {X 0,Y 472.318,Z 667.131,A -85,B 0,C 180,E1 12231.294,E2 12231.294} C_VEL
LIN {X 0,Y 474.849,Z 672.034,A -85,B 0,C 180,E1 12229.137,E2 12229.137} C_VEL
LIN {X 0,Y 475.349,Z 673.141,A -85,B 0,C 180,E1 12228.751,E2 12228.751} C_VEL
LIN {X 0,Y 454.141,Z 886.693,A -85,B 0,C 180,E1 12225.633,E2 12225.633} C_VEL
LIN {X 0,Y 450.979,Z 909.945,A -85,B 0,C 180,E1 12225.255,E2 12225.255} C_VEL
LIN {X 0,Y 446.844,Z 932.147,A -85,B 0,C 180,E1 12224.852,E2 12224.852} C_VEL
LIN {X 0,Y 441.082,Z 956.667,A -85,B 0,C 180,E1 12224.317,E2 12224.317} C_VEL
LIN {X 0,Y 433.124,Z 983.859,A -85,B 0,C 180,E1 12223.545,E2 12223.545} C_VEL
LIN {X 0,Y 425.739,Z 1005.288,A -85,B 0,C 180,E1 12222.787,E2 12222.787} C_VEL
LIN {X 0,Y 418.051,Z 1025.051,A -85,B 0,C 180,E1 12221.95,E2 12221.95} C_VEL
LIN {X 0,Y 409.393,Z 1045.018,A -85,B 0,C 180,E1 12220.953,E2 12220.953} C_VEL
LIN {X 0,Y 398.414,Z 1067.916,A -85,B 0,C 180,E1 12219.583,E2 12219.583} C_VEL
LIN {X 0,Y 385.855,Z 1091.057,A -85,B 0,C 180,E1 12217.892,E2 12217.892} C_VEL
LIN {X 0,Y 375.114,Z 1109.23,A -85,B 0,C 180,E1 12216.303,E2 12216.303} C_VEL
LIN {X 0,Y 364.332,Z 1126.243,A -85,B 0,C 180,E1 12214.555,E2 12214.555} C_VEL
LIN {X 0,Y 352.851,Z 1143.227,A -85,B 0,C 180,E1 12212.503,E2 12212.503} C_VEL
LIN {X 0,Y 337.842,Z 1163.96,A -85,B 0,C 180,E1 12209.467,E2 12209.467} C_VEL
LIN {X 0,Y 325.909,Z 1179.456,A -85,B 0,C 180,E1 12206.69,E2 12206.69} C_VEL
LIN {X 0,Y 315.214,Z 1192.852,A -85,B 0,C 180,E1 12203.842,E2 12203.842} C_VEL
LIN {X 0,Y 304.432,Z 1205.998,A -85,B 0,C 180,E1 12200.529,E2 12200.529} C_VEL
LIN {X 0,Y 292.079,Z 1220.847,A -85,B 0,C 180,E1 12195.974,E2 12195.974} C_VEL
LIN {X 0,Y 282.309,Z 1232.556,A -85,B 0,C 180,E1 12191.486,E2 12191.486} C_VEL
LIN {X 0,Y 275.084,Z 1241.482,A -85,B 0,C 180,E1 12187.384,E2 12187.384} C_VEL
LIN {X 0,Y 268.835,Z 1249.633,A -85,B 0,C 180,E1 12182.899,E2 12182.899} C_VEL
LIN {X 0,Y 263.543,Z 1257.224,A -85,B 0,C 180,E1 12177.827,E2 12177.827} C_VEL
LIN {X 0,Y 259.195,Z 1264.572,A -85,B 0,C 180,E1 12171.508,E2 12171.508} C_VEL
LIN {X 0,Y 257.201,Z 1268.969,A -85,B 0,C 180,E1 12166.496,E2 12166.496} C_VEL
LIN {X 0,Y 256.317,Z 1271.971,A -85,B 0,C 180,E1 12161.942,E2 12161.942} C_VEL
LIN {X 0,Y 256.017,Z 1274.019,A -85,B 0,C 180,E1 12157.415,E2 12157.415} C_VEL
LIN {X 0,Y 255.998,Z 1275.092,A -85,B 0,C 180,E1 12153.145,E2 12153.145} C_VEL
LIN {X 0,Y 255.983,Z 1275.307,A -85,B 0,C 180,E1 12148.891,E2 12148.891} C_VEL
LIN {X 0,Y 255.997,Z 1274.593,A -85,B 0,C 180,E1 12144.407,E2 12144.407} C_VEL
LIN {X 0,Y 256.135,Z 1272.801,A -85,B 0,C 180,E1 12139.658,E2 12139.658} C_VEL
LIN {X 0,Y 256.864,Z 1269.962,A -85,B 0,C 180,E1 12134.882,E2 12134.882} C_VEL
LIN {X 0,Y 258.45,Z 1266.046,A -85,B 0,C 180,E1 12130.072,E2 12130.072} C_VEL
LIN {X 0,Y 261.077,Z 1261.106,A -85,B 0,C 180,E1 12125.339,E2 12125.339} C_VEL
LIN {X 0,Y 264.913,Z 1255.091,A -85,B 0,C 180,E1 12120.679,E2 12120.679} C_VEL
LIN {X 0,Y 270.441,Z 1247.44,A -85,B 0,C 180,E1 12115.821,E2 12115.821} C_VEL
LIN {X 0,Y 279.605,Z 1235.815,A -85,B 0,C 180,E1 12109.932,E2 12109.932} C_VEL
LIN {X 0,Y 288.466,Z 1225.053,A -85,B 0,C 180,E1 12105.575,E2 12105.575} C_VEL
LIN {X 0,Y 297.266,Z 1214.518,A -85,B 0,C 180,E1 12101.998,E2 12101.998} C_VEL
LIN {X 0,Y 307.587,Z 1202.09,A -85,B 0,C 180,E1 12098.442,E2 12098.442} C_VEL
LIN {X 0,Y 321.185,Z 1185.383,A -85,B 0,C 180,E1 12094.513,E2 12094.513} C_VEL
LIN {X 0,Y 333.838,Z 1169.049,A -85,B 0,C 180,E1 12091.41,E2 12091.41} C_VEL
LIN {X 0,Y 345.137,Z 1153.843,A -85,B 0,C 180,E1 12088.987,E2 12088.987} C_VEL
LIN {X 0,Y 356.661,Z 1137.515,A -85,B 0,C 180,E1 12086.782,E2 12086.782} C_VEL
LIN {X 0,Y 370.577,Z 1116.453,A -85,B 0,C 180,E1 12084.412,E2 12084.412} C_VEL
LIN {X 0,Y 383.064,Z 1095.663,A -85,B 0,C 180,E1 12082.504,E2 12082.504} C_VEL
LIN {X 0,Y 392.957,Z 1077.869,A -85,B 0,C 180,E1 12081.121,E2 12081.121} C_VEL
LIN {X 0,Y 402.8,Z 1058.614,A -85,B 0,C 180,E1 12079.841,E2 12079.841} C_VEL
LIN {X 0,Y 413.001,Z 1036.702,A -85,B 0,C 180,E1 12078.618,E2 12078.618} C_VEL
LIN {X 0,Y 423.43,Z 1011.077,A -85,B 0,C 180,E1 12077.452,E2 12077.452} C_VEL
LIN {X 0,Y 430.977,Z 989.825,A -85,B 0,C 180,E1 12076.661,E2 12076.661} C_VEL
LIN {X 0,Y 437.245,Z 969.691,A -85,B 0,C 180,E1 12076.038,E2 12076.038} C_VEL
LIN {X 0,Y 442.951,Z 948.372,A -85,B 0,C 180,E1 12075.495,E2 12075.495} C_VEL
LIN {X 0,Y 448.253,Z 924.46,A -85,B 0,C 180,E1 12075.008,E2 12075.008} C_VEL
LIN {X 0,Y 452.982,Z 894.861,A -85,B 0,C 180,E1 12074.501,E2 12074.501} C_VEL
LIN {X 0,Y 459.867,Z 826.99,A -85,B 0,C 180,E1 12073.492,E2 12073.492} C_VEL
LIN {X 0,Y 475.139,Z 672.818,A -85,B 0,C 180,E1 12071.231,E2 12071.231} C_VEL
LIN {X 0,Y 472.36,Z 667.508,A -85,B 0,C 180,E1 12068.951,E2 12068.951} C_VEL
LIN {X 0,Y 471.075,Z 665.204,A -85,B 0,C 180,E1 12067.685,E2 12067.685} C_VEL
LIN {X 0,Y 469.355,Z 661.715,A -85,B 0,C 180,E1 12065.501,E2 12065.501} C_VEL
LIN {X 0,Y 467.698,Z 657.93,A -85,B 0,C 180,E1 12061.593,E2 12061.593} C_VEL
LIN {X 0,Y 467.612,Z 657.216,A -85,B 0,C 180,E1 12060.735,E2 12060.735} C_VEL
LIN {X 0,Y 467.656,Z 657.329,A -85,B 0,C 180,E1 12058.407,E2 12058.407} C_VEL
LIN {X 0,Y 469.346,Z 661.686,A -85,B 0,C 180,E1 12054.008,E2 12054.008} C_VEL
LIN {X 0,Y 472.028,Z 666.85,A -85,B 0,C 180,E1 12050.859,E2 12050.859} C_VEL
LIN {X 0,Y 474.713,Z 672.006,A -85,B 0,C 180,E1 12048.58,E2 12048.58} C_VEL
LIN {X 0,Y 475.001,Z 672.79,A -85,B 0,C 180,E1 12048.347,E2 12048.347} C_VEL
LIN {X 0,Y 453.907,Z 883.737,A -85,B 0,C 180,E1 12045.27,E2 12045.27} C_VEL
LIN {X 0,Y 450.578,Z 906.663,A -85,B 0,C 180,E1 12044.893,E2 12044.893} C_VEL
LIN {X 0,Y 445.048,Z 934.578,A -85,B 0,C 180,E1 12044.315,E2 12044.315} C_VEL
LIN {X 0,Y 438.841,Z 958.715,A -85,B 0,C 180,E1 12043.668,E2 12043.668} C_VEL
LIN {X 0,Y 432.768,Z 978.8,A -85,B 0,C 180,E1 12043.012,E2 12043.012} C_VEL
LIN {X 0,Y 426.127,Z 998.024,A -85,B 0,C 180,E1 12042.269,E2 12042.269} C_VEL
LIN {X 0,Y 418.321,Z 1018.036,A -85,B 0,C 180,E1 12041.364,E2 12041.364} C_VEL
LIN {X 0,Y 408.624,Z 1040.231,A -85,B 0,C 180,E1 12040.168,E2 12040.168} C_VEL
LIN {X 0,Y 396.677,Z 1064.225,A -85,B 0,C 180,E1 12038.604,E2 12038.604} C_VEL
LIN {X 0,Y 386.263,Z 1083.098,A -85,B 0,C 180,E1 12037.128,E2 12037.128} C_VEL
LIN {X 0,Y 376.074,Z 1100.152,A -85,B 0,C 180,E1 12035.568,E2 12035.568} C_VEL
LIN {X 0,Y 365.427,Z 1116.705,A -85,B 0,C 180,E1 12033.806,E2 12033.806} C_VEL
LIN {X 0,Y 352.017,Z 1136.195,A -85,B 0,C 180,E1 12031.344,E2 12031.344} C_VEL
LIN {X 0,Y 338.589,Z 1154.058,A -85,B 0,C 180,E1 12028.568,E2 12028.568} C_VEL
LIN {X 0,Y 327.803,Z 1167.705,A -85,B 0,C 180,E1 12026.046,E2 12026.046} C_VEL
LIN {X 0,Y 316.971,Z 1180.856,A -85,B 0,C 180,E1 12023.176,E2 12023.176} C_VEL
LIN {X 0,Y 306.059,Z 1193.685,A -85,B 0,C 180,E1 12019.843,E2 12019.843} C_VEL
LIN {X 0,Y 293.007,Z 1208.597,A -85,B 0,C 180,E1 12015.058,E2 12015.058} C_VEL
LIN {X 0,Y 283.834,Z 1218.951,A -85,B 0,C 180,E1 12010.923,E2 12010.923} C_VEL
LIN {X 0,Y 276.54,Z 1227.373,A -85,B 0,C 180,E1 12006.871,E2 12006.871} C_VEL
LIN {X 0,Y 269.874,Z 1235.367,A -85,B 0,C 180,E1 12002.23,E2 12002.23} C_VEL
LIN {X 0,Y 263.469,Z 1243.726,A -85,B 0,C 180,E1 11996.106,E2 11996.106} C_VEL
LIN {X 0,Y 259.723,Z 1249.3,A -85,B 0,C 180,E1 11990.688,E2 11990.688} C_VEL
LIN {X 0,Y 257.688,Z 1253.031,A -85,B 0,C 180,E1 11985.98,E2 11985.98} C_VEL
LIN {X 0,Y 256.609,Z 1255.689,A -85,B 0,C 180,E1 11981.451,E2 11981.451} C_VEL
LIN {X 0,Y 256.171,Z 1257.398,A -85,B 0,C 180,E1 11977.164,E2 11977.164} C_VEL
LIN {X 0,Y 256.025,Z 1258.328,A -85,B 0,C 180,E1 11972.9,E2 11972.9} C_VEL
LIN {X 0,Y 255.995,Z 1258.488,A -85,B 0,C 180,E1 11968.647,E2 11968.647} C_VEL
LIN {X 0,Y 256.098,Z 1257.814,A -85,B 0,C 180,E1 11964.164,E2 11964.164} C_VEL
LIN {X 0,Y 256.418,Z 1256.278,A -85,B 0,C 180,E1 11959.657,E2 11959.657} C_VEL
LIN {X 0,Y 257.407,Z 1253.706,A -85,B 0,C 180,E1 11954.905,E2 11954.905} C_VEL
LIN {X 0,Y 259.239,Z 1250.138,A -85,B 0,C 180,E1 11950.149,E2 11950.149} C_VEL
LIN {X 0,Y 262.149,Z 1245.542,A -85,B 0,C 180,E1 11945.424,E2 11945.424} C_VEL
LIN {X 0,Y 266.085,Z 1240.172,A -85,B 0,C 180,E1 11940.994,E2 11940.994} C_VEL
LIN {X 0,Y 271.729,Z 1233.144,A -85,B 0,C 180,E1 11936.266,E2 11936.266} C_VEL
LIN {X 0,Y 280.341,Z 1223.144,A -85,B 0,C 180,E1 11930.844,E2 11930.844} C_VEL
LIN {X 0,Y 290.082,Z 1211.949,A -85,B 0,C 180,E1 11926.088,E2 11926.088} C_VEL
LIN {X 0,Y 299.308,Z 1201.468,A -85,B 0,C 180,E1 11922.405,E2 11922.405} C_VEL
LIN {X 0,Y 309.147,Z 1190.171,A -85,B 0,C 180,E1 11919.073,E2 11919.073} C_VEL
LIN {X 0,Y 321.658,Z 1175.47,A -85,B 0,C 180,E1 11915.459,E2 11915.459} C_VEL
LIN {X 0,Y 335.248,Z 1158.509,A -85,B 0,C 180,E1 11912.1,E2 11912.1} C_VEL
LIN {X 0,Y 346.436,Z 1143.827,A -85,B 0,C 180,E1 11909.677,E2 11909.677} C_VEL
LIN {X 0,Y 357.467,Z 1128.532,A -85,B 0,C 180,E1 11907.53,E2 11907.53} C_VEL
LIN {X 0,Y 369.434,Z 1110.866,A -85,B 0,C 180,E1 11905.428,E2 11905.428} C_VEL
LIN {X 0,Y 383.698,Z 1087.821,A -85,B 0,C 180,E1 11903.172,E2 11903.172} C_VEL
LIN {X 0,Y 394.292,Z 1068.987,A -85,B 0,C 180,E1 11901.647,E2 11901.647} C_VEL
LIN {X 0,Y 403.352,Z 1051.45,A -85,B 0,C 180,E1 11900.43,E2 11900.43} C_VEL
LIN {X 0,Y 412.153,Z 1032.748,A -85,B 0,C 180,E1 11899.305,E2 11899.305} C_VEL
LIN {X 0,Y 421.117,Z 1011.656,A -85,B 0,C 180,E1 11898.231,E2 11898.231} C_VEL
LIN {X 0,Y 431.036,Z 984.678,A -85,B 0,C 180,E1 11897.103,E2 11897.103} C_VEL
LIN {X 0,Y 437.727,Z 963.272,A -85,B 0,C 180,E1 11896.374,E2 11896.374} C_VEL
LIN {X 0,Y 440.585,Z 953.296,A -85,B 0,C 180,E1 11896.074,E2 11896.074} C_VEL
LIN {X 0,Y 442.269,Z 946.137,A -85,B 0,C 180,E1 11895.749,E2 11895.749} C_VEL
LIN {X 0,Y 444.814,Z 928.394,A -85,B 0,C 180,E1 11894.568,E2 11894.568} C_VEL
LIN {X 0,Y 446.079,Z 921.065,A -85,B 0,C 180,E1 11894.289,E2 11894.289} C_VEL
LIN {X 0,Y 450.579,Z 895.95,A -85,B 0,C 180,E1 11893.837,E2 11893.837} C_VEL
LIN {X 0,Y 454.837,Z 859.034,A -85,B 0,C 180,E1 11893.281,E2 11893.281} C_VEL
LIN {X 0,Y 473.077,Z 678.758,A -85,B 0,C 180,E1 11890.688,E2 11890.688} C_VEL
LIN {X 0,Y 470.274,Z 673.282,A -85,B 0,C 180,E1 11888.067,E2 11888.067} C_VEL
LIN {X 0,Y 468.415,Z 669.554,A -85,B 0,C 180,E1 11885.635,E2 11885.635} C_VEL
LIN {X 0,Y 466.91,Z 665.468,A -85,B 0,C 180,E1 11881.35,E2 11881.35} C_VEL
LIN {X 0,Y 466.864,Z 665.207,A -85,B 0,C 180,E1 11879.755,E2 11879.755} C_VEL
LIN {X 0,Y 466.918,Z 665.645,A -85,B 0,C 180,E1 11878.896,E2 11878.896} C_VEL
LIN {X 0,Y 468.529,Z 669.712,A -85,B 0,C 180,E1 11874.612,E2 11874.612} C_VEL
LIN {X 0,Y 471.139,Z 674.951,A -85,B 0,C 180,E1 11871.456,E2 11871.456} C_VEL
LIN {X 0,Y 473.208,Z 679.07,A -85,B 0,C 180,E1 11869.618,E2 11869.618} C_VEL
LIN {X 0,Y 451.945,Z 888.648,A -85,B 0,C 180,E1 11866.588,E2 11866.588} C_VEL
LIN {X 0,Y 448.774,Z 911.047,A -85,B 0,C 180,E1 11866.226,E2 11866.226} C_VEL
LIN {X 0,Y 444.332,Z 934.167,A -85,B 0,C 180,E1 11865.811,E2 11865.811} C_VEL
LIN {X 0,Y 437.253,Z 962.671,A -85,B 0,C 180,E1 11865.174,E2 11865.174} C_VEL
LIN {X 0,Y 430.248,Z 985.541,A -85,B 0,C 180,E1 11864.516,E2 11864.516} C_VEL
LIN {X 0,Y 422.812,Z 1006.604,A -85,B 0,C 180,E1 11863.777,E2 11863.777} C_VEL
LIN {X 0,Y 414.643,Z 1027.078,A -85,B 0,C 180,E1 11862.916,E2 11862.916} C_VEL
LIN {X 0,Y 403.901,Z 1051.102,A -85,B 0,C 180,E1 11861.703,E2 11861.703} C_VEL
LIN {X 0,Y 392.044,Z 1074.277,A -85,B 0,C 180,E1 11860.25,E2 11860.25} C_VEL
LIN {X 0,Y 381.633,Z 1092.812,A -85,B 0,C 180,E1 11858.875,E2 11858.875} C_VEL
LIN {X 0,Y 370.702,Z 1110.805,A -85,B 0,C 180,E1 11857.301,E2 11857.301} C_VEL
LIN {X 0,Y 358.337,Z 1129.726,A -85,B 0,C 180,E1 11855.336,E2 11855.336} C_VEL
LIN {X 0,Y 343.346,Z 1150.811,A -85,B 0,C 180,E1 11852.66,E2 11852.66} C_VEL
LIN {X 0,Y 331.62,Z 1166.26,A -85,B 0,C 180,E1 11850.28,E2 11850.28} C_VEL
LIN {X 0,Y 320.492,Z 1180.251,A -85,B 0,C 180,E1 11847.733,E2 11847.733} C_VEL
LIN {X 0,Y 309.418,Z 1193.646,A -85,B 0,C 180,E1 11844.852,E2 11844.852} C_VEL
LIN {X 0,Y 296.427,Z 1208.959,A -85,B 0,C 180,E1 11840.889,E2 11840.889} C_VEL
LIN {X 0,Y 284.369,Z 1222.678,A -85,B 0,C 180,E1 11836.423,E2 11836.423} C_VEL
LIN {X 0,Y 275.629,Z 1232.751,A -85,B 0,C 180,E1 11832.444,E2 11832.444} C_VEL
LIN {X 0,Y 268.086,Z 1241.623,A -85,B 0,C 180,E1 11828.263,E2 11828.263} C_VEL
LIN {X 0,Y 261.532,Z 1249.722,A -85,B 0,C 180,E1 11823.677,E2 11823.677} C_VEL
LIN {X 0,Y 255.355,Z 1258.222,A -85,B 0,C 180,E1 11817.755,E2 11817.755} C_VEL
LIN {X 0,Y 251.259,Z 1264.732,A -85,B 0,C 180,E1 11811.731,E2 11811.731} C_VEL
LIN {X 0,Y 249.273,Z 1268.867,A -85,B 0,C 180,E1 11806.797,E2 11806.797} C_VEL
LIN {X 0,Y 248.333,Z 1271.824,A -85,B 0,C 180,E1 11802.096,E2 11802.096} C_VEL
LIN {X 0,Y 248.02,Z 1273.827,A -85,B 0,C 180,E1 11797.422,E2 11797.422} C_VEL
LIN {X 0,Y 248.001,Z 1274.829,A -85,B 0,C 180,E1 11793.246,E2 11793.246} C_VEL
LIN {X 0,Y 247.988,Z 1275.044,A -85,B 0,C 180,E1 11788.855,E2 11788.855} C_VEL
LIN {X 0,Y 248.001,Z 1274.329,A -85,B 0,C 180,E1 11784.226,E2 11784.226} C_VEL
LIN {X 0,Y 248.168,Z 1272.539,A -85,B 0,C 180,E1 11779.331,E2 11779.331} C_VEL
LIN {X 0,Y 248.958,Z 1269.701,A -85,B 0,C 180,E1 11774.402,E2 11774.402} C_VEL
LIN {X 0,Y 250.673,Z 1265.806,A -85,B 0,C 180,E1 11769.463,E2 11769.463} C_VEL
LIN {X 0,Y 253.547,Z 1260.832,A -85,B 0,C 180,E1 11764.555,E2 11764.555} C_VEL
LIN {X 0,Y 257.695,Z 1254.751,A -85,B 0,C 180,E1 11759.721,E2 11759.721} C_VEL
LIN {X 0,Y 263.842,Z 1246.786,A -85,B 0,C 180,E1 11754.567,E2 11754.567} C_VEL
LIN {X 0,Y 273.57,Z 1235.092,A -85,B 0,C 180,E1 11748.598,E2 11748.598} C_VEL
LIN {X 0,Y 282.485,Z 1224.774,A -85,B 0,C 180,E1 11744.373,E2 11744.373} C_VEL
LIN {X 0,Y 291.67,Z 1214.238,A -85,B 0,C 180,E1 11740.763,E2 11740.763} C_VEL
LIN {X 0,Y 302.402,Z 1201.811,A -85,B 0,C 180,E1 11737.187,E2 11737.187} C_VEL
LIN {X 0,Y 316.021,Z 1185.689,A -85,B 0,C 180,E1 11733.374,E2 11733.374} C_VEL
LIN {X 0,Y 329.529,Z 1168.78,A -85,B 0,C 180,E1 11730.165,E2 11730.165} C_VEL
LIN {X 0,Y 341.154,Z 1153.565,A -85,B 0,C 180,E1 11727.755,E2 11727.755} C_VEL
LIN {X 0,Y 352.974,Z 1137.238,A -85,B 0,C 180,E1 11725.571,E2 11725.571} C_VEL
LIN {X 0,Y 366.95,Z 1116.611,A -85,B 0,C 180,E1 11723.273,E2 11723.273} C_VEL
LIN {X 0,Y 379.971,Z 1095.387,A -85,B 0,C 180,E1 11721.35,E2 11721.35} C_VEL
LIN {X 0,Y 389.932,Z 1077.84,A -85,B 0,C 180,E1 11720.01,E2 11720.01} C_VEL
LIN {X 0,Y 399.84,Z 1058.834,A -85,B 0,C 180,E1 11718.765,E2 11718.765} C_VEL
LIN {X 0,Y 409.782,Z 1037.902,A -85,B 0,C 180,E1 11717.612,E2 11717.612} C_VEL
LIN {X 0,Y 421.015,Z 1010.926,A -85,B 0,C 180,E1 11716.4,E2 11716.4} C_VEL
LIN {X 0,Y 428.722,Z 989.551,A -85,B 0,C 180,E1 11715.622,E2 11715.622} C_VEL
LIN {X 0,Y 435.416,Z 968.268,A -85,B 0,C 180,E1 11714.983,E2 11714.983} C_VEL
LIN {X 0,Y 441.287,Z 946.432,A -85,B 0,C 180,E1 11714.449,E2 11714.449} C_VEL
LIN {X 0,Y 447.285,Z 918.889,A -85,B 0,C 180,E1 11713.913,E2 11713.913} C_VEL
LIN {X 0,Y 451.278,Z 892.534,A -85,B 0,C 180,E1 11713.479,E2 11713.479} C_VEL
LIN {X 0,Y 467.806,Z 729.81,A -85,B 0,C 180,E1 11711.114,E2 11711.114} C_VEL
LIN {X 0,Y 472.983,Z 678.925,A -85,B 0,C 180,E1 11710.37,E2 11710.37} C_VEL
LIN {X 0,Y 470.455,Z 673.792,A -85,B 0,C 180,E1 11708.064,E2 11708.064} C_VEL
LIN {X 0,Y 468.208,Z 669.497,A -85,B 0,C 180,E1 11705.269,E2 11705.269} C_VEL
LIN {X 0,Y 466.699,Z 665.81,A -85,B 0,C 180,E1 11701.473,E2 11701.473} C_VEL
LIN {X 0,Y 466.621,Z 665.161,A -85,B 0,C 180,E1 11700.614,E2 11700.614} C_VEL
LIN {X 0,Y 466.67,Z 665.367,A -85,B 0,C 180,E1 11698.404,E2 11698.404} C_VEL
LIN {X 0,Y 468.61,Z 670.248,A -85,B 0,C 180,E1 11693.63,E2 11693.63} C_VEL
LIN {X 0,Y 470.909,Z 674.809,A -85,B 0,C 180,E1 11690.96,E2 11690.96} C_VEL
LIN {X 0,Y 472.871,Z 678.679,A -85,B 0,C 180,E1 11689.216,E2 11689.216} C_VEL
LIN {X 0,Y 451.873,Z 884.556,A -85,B 0,C 180,E1 11686.244,E2 11686.244} C_VEL
LIN {X 0,Y 448.344,Z 908.238,A -85,B 0,C 180,E1 11685.858,E2 11685.858} C_VEL
LIN {X 0,Y 442.27,Z 937.552,A -85,B 0,C 180,E1 11685.25,E2 11685.25} C_VEL
LIN {X 0,Y 436.435,Z 959.724,A -85,B 0,C 180,E1 11684.658,E2 11684.658} C_VEL
LIN {X 0,Y 430.061,Z 980.35,A -85,B 0,C 180,E1 11683.992,E2 11683.992} C_VEL
LIN {X 0,Y 422.901,Z 1000.543,A -85,B 0,C 180,E1 11683.216,E2 11683.216} C_VEL
LIN {X 0,Y 413.341,Z 1024.27,A -85,B 0,C 180,E1 11682.13,E2 11682.13} C_VEL
LIN {X 0,Y 402.284,Z 1047.992,A -85,B 0,C 180,E1 11680.792,E2 11680.792} C_VEL
LIN {X 0,Y 392.227,Z 1067.329,A -85,B 0,C 180,E1 11679.502,E2 11679.502} C_VEL
LIN {X 0,Y 381.99,Z 1085.354,A -85,B 0,C 180,E1 11678.088,E2 11678.088} C_VEL
LIN {X 0,Y 370.858,Z 1103.434,A -85,B 0,C 180,E1 11676.422,E2 11676.422} C_VEL
LIN {X 0,Y 356.478,Z 1124.828,A -85,B 0,C 180,E1 11674.051,E2 11674.051} C_VEL
LIN {X 0,Y 343.913,Z 1141.964,A -85,B 0,C 180,E1 11671.734,E2 11671.734} C_VEL
LIN {X 0,Y 333.006,Z 1155.997,A -85,B 0,C 180,E1 11669.493,E2 11669.493} C_VEL
LIN {X 0,Y 321.973,Z 1169.495,A -85,B 0,C 180,E1 11666.961,E2 11666.961} C_VEL
LIN {X 0,Y 309.99,Z 1183.543,A -85,B 0,C 180,E1 11663.823,E2 11663.823} C_VEL
LIN {X 0,Y 295.936,Z 1199.297,A -85,B 0,C 180,E1 11659.466,E2 11659.466} C_VEL
LIN {X 0,Y 285.526,Z 1210.622,A -85,B 0,C 180,E1 11655.577,E2 11655.577} C_VEL
LIN {X 0,Y 276.761,Z 1220.121,A -85,B 0,C 180,E1 11651.648,E2 11651.648} C_VEL
LIN {X 0,Y 268.523,Z 1229.224,A -85,B 0,C 180,E1 11647.087,E2 11647.087} C_VEL
LIN {X 0,Y 260.155,Z 1238.862,A -85,B 0,C 180,E1 11640.985,E2 11640.985} C_VEL
LIN {X 0,Y 255.084,Z 1245.224,A -85,B 0,C 180,E1 11635.779,E2 11635.779} C_VEL
LIN {X 0,Y 251.818,Z 1249.93,A -85,B 0,C 180,E1 11630.926,E2 11630.926} C_VEL
LIN {X 0,Y 249.772,Z 1253.452,A -85,B 0,C 180,E1 11626.262,E2 11626.262} C_VEL
LIN {X 0,Y 248.638,Z 1256.063,A -85,B 0,C 180,E1 11621.588,E2 11621.588} C_VEL
LIN {X 0,Y 248.177,Z 1257.726,A -85,B 0,C 180,E1 11617.164,E2 11617.164} C_VEL
LIN {X 0,Y 248.03,Z 1258.591,A -85,B 0,C 180,E1 11612.993,E2 11612.993} C_VEL
LIN {X 0,Y 248.001,Z 1258.751,A -85,B 0,C 180,E1 11608.603,E2 11608.603} C_VEL
LIN {X 0,Y 248.112,Z 1258.077,A -85,B 0,C 180,E1 11603.975,E2 11603.975} C_VEL
LIN {X 0,Y 248.466,Z 1256.543,A -85,B 0,C 180,E1 11599.322,E2 11599.322} C_VEL
LIN {X 0,Y 249.548,Z 1253.973,A -85,B 0,C 180,E1 11594.418,E2 11594.418} C_VEL
LIN {X 0,Y 251.537,Z 1250.407,A -85,B 0,C 180,E1 11589.514,E2 11589.514} C_VEL
LIN {X 0,Y 254.664,Z 1245.812,A -85,B 0,C 180,E1 11584.652,E2 11584.652} C_VEL
LIN {X 0,Y 258.857,Z 1240.443,A -85,B 0,C 180,E1 11580.103,E2 11580.103} C_VEL
LIN {X 0,Y 264.576,Z 1233.719,A -85,B 0,C 180,E1 11575.457,E2 11575.457} C_VEL
LIN {X 0,Y 273.152,Z 1224.25,A -85,B 0,C 180,E1 11570.154,E2 11570.154} C_VEL
LIN {X 0,Y 283.667,Z 1212.724,A -85,B 0,C 180,E1 11565.113,E2 11565.113} C_VEL
LIN {X 0,Y 293.233,Z 1202.301,A -85,B 0,C 180,E1 11561.385,E2 11561.385} C_VEL
LIN {X 0,Y 303.401,Z 1191.065,A -85,B 0,C 180,E1 11558.024,E2 11558.024} C_VEL
LIN {X 0,Y 314.456,Z 1178.494,A -85,B 0,C 180,E1 11554.868,E2 11554.868} C_VEL
LIN {X 0,Y 329.001,Z 1161.206,A -85,B 0,C 180,E1 11551.312,E2 11551.312} C_VEL
LIN {X 0,Y 341.726,Z 1145.008,A -85,B 0,C 180,E1 11548.612,E2 11548.612} C_VEL
LIN {X 0,Y 353.01,Z 1129.8,A -85,B 0,C 180,E1 11546.474,E2 11546.474} C_VEL
LIN {X 0,Y 364.367,Z 1113.498,A -85,B 0,C 180,E1 11544.527,E2 11544.527} C_VEL
LIN {X 0,Y 377.27,Z 1093.595,A -85,B 0,C 180,E1 11542.526,E2 11542.526} C_VEL
LIN {X 0,Y 390.479,Z 1070.861,A -85,B 0,C 180,E1 11540.656,E2 11540.656} C_VEL
LIN {X 0,Y 400.181,Z 1052.517,A -85,B 0,C 180,E1 11539.391,E2 11539.391} C_VEL
LIN {X 0,Y 409.133,Z 1033.902,A -85,B 0,C 180,E1 11538.283,E2 11538.283} C_VEL
LIN {X 0,Y 417.978,Z 1013.538,A -85,B 0,C 180,E1 11537.256,E2 11537.256} C_VEL
LIN {X 0,Y 427.475,Z 988.766,A -85,B 0,C 180,E1 11536.212,E2 11536.212} C_VEL
LIN {X 0,Y 435.316,Z 964.263,A -85,B 0,C 180,E1 11535.381,E2 11535.381} C_VEL
LIN {X 0,Y 441.22,Z 942.542,A -85,B 0,C 180,E1 11534.776,E2 11534.776} C_VEL
LIN {X 0,Y 446.079,Z 921.065,A -85,B 0,C 180,E1 11534.289,E2 11534.289} C_VEL
LIN {X 0,Y 447.398,Z 913.688,A -85,B 0,C 180,E1 11534.026,E2 11534.026} C_VEL
LIN {X 0,Y 449.211,Z 894.395,A -85,B 0,C 180,E1 11532.916,E2 11532.916} C_VEL
LIN {X 0,Y 449.859,Z 887.957,A -85,B 0,C 180,E1 11532.717,E2 11532.717} C_VEL
LIN {X 0,Y 456.882,Z 821.729,A -85,B 0,C 180,E1 11531.758,E2 11531.758} C_VEL
LIN {X 0,Y 471.038,Z 684.847,A -85,B 0,C 180,E1 11529.811,E2 11529.811} C_VEL
LIN {X 0,Y 469.067,Z 680.994,A -85,B 0,C 180,E1 11527.841,E2 11527.841} C_VEL
LIN {X 0,Y 467.358,Z 677.437,A -85,B 0,C 180,E1 11525.525,E2 11525.525} C_VEL
LIN {X 0,Y 465.924,Z 673.205,A -85,B 0,C 180,E1 11521.107,E2 11521.107} C_VEL
LIN {X 0,Y 465.927,Z 673.381,A -85,B 0,C 180,E1 11519.139,E2 11519.139} C_VEL
LIN {X 0,Y 467.386,Z 677.501,A -85,B 0,C 180,E1 11514.845,E2 11514.845} C_VEL
LIN {X 0,Y 469.905,Z 682.639,A -85,B 0,C 180,E1 11511.68,E2 11511.68} C_VEL
LIN {X 0,Y 471.148,Z 685.275,A -85,B 0,C 180,E1 11510.489,E2 11510.489} C_VEL
LIN {X 0,Y 449.844,Z 890.86,A -85,B 0,C 180,E1 11507.547,E2 11507.547} C_VEL
LIN {X 0,Y 446.383,Z 914.04,A -85,B 0,C 180,E1 11507.175,E2 11507.175} C_VEL
LIN {X 0,Y 440.332,Z 943.077,A -85,B 0,C 180,E1 11506.642,E2 11506.642} C_VEL
LIN {X 0,Y 433.952,Z 966.784,A -85,B 0,C 180,E1 11506.089,E2 11506.089} C_VEL
LIN {X 0,Y 427.58,Z 986.98,A -85,B 0,C 180,E1 11505.508,E2 11505.508} C_VEL
LIN {X 0,Y 420.181,Z 1007.481,A -85,B 0,C 180,E1 11504.798,E2 11504.798} C_VEL
LIN {X 0,Y 411.588,Z 1028.552,A -85,B 0,C 180,E1 11503.922,E2 11503.922} C_VEL
LIN {X 0,Y 399.299,Z 1054.962,A -85,B 0,C 180,E1 11502.578,E2 11502.578} C_VEL
LIN {X 0,Y 388.516,Z 1075.493,A -85,B 0,C 180,E1 11501.289,E2 11501.289} C_VEL
LIN {X 0,Y 378.329,Z 1093.219,A -85,B 0,C 180,E1 11499.988,E2 11499.988} C_VEL
LIN {X 0,Y 367.133,Z 1111.238,A -85,B 0,C 180,E1 11498.428,E2 11498.428} C_VEL
LIN {X 0,Y 353.453,Z 1131.664,A -85,B 0,C 180,E1 11496.315,E2 11496.315} C_VEL
LIN {X 0,Y 338.86,Z 1151.478,A -85,B 0,C 180,E1 11493.781,E2 11493.781} C_VEL
LIN {X 0,Y 326.849,Z 1166.845,A -85,B 0,C 180,E1 11491.411,E2 11491.411} C_VEL
LIN {X 0,Y 315.425,Z 1180.761,A -85,B 0,C 180,E1 11488.869,E2 11488.869} C_VEL
LIN {X 0,Y 303.416,Z 1194.797,A -85,B 0,C 180,E1 11485.818,E2 11485.818} C_VEL
LIN {X 0,Y 288.411,Z 1211.638,A -85,B 0,C 180,E1 11481.276,E2 11481.276} C_VEL
LIN {X 0,Y 277.633,Z 1223.455,A -85,B 0,C 180,E1 11477.292,E2 11477.292} C_VEL
LIN {X 0,Y 268.602,Z 1233.416,A -85,B 0,C 180,E1 11473.242,E2 11473.242} C_VEL
LIN {X 0,Y 260.083,Z 1243.013,A -85,B 0,C 180,E1 11468.532,E2 11468.532} C_VEL
LIN {X 0,Y 251.452,Z 1253.339,A -85,B 0,C 180,E1 11462.114,E2 11462.114} C_VEL
LIN {X 0,Y 246.442,Z 1260.035,A -85,B 0,C 180,E1 11456.777,E2 11456.777} C_VEL
LIN {X 0,Y 243.173,Z 1265.151,A -85,B 0,C 180,E1 11451.677,E2 11451.677} C_VEL
LIN {X 0,Y 241.249,Z 1268.997,A -85,B 0,C 180,E1 11446.781,E2 11446.781} C_VEL
LIN {X 0,Y 240.321,Z 1271.797,A -85,B 0,C 180,E1 11442.017,E2 11442.017} C_VEL
LIN {X 0,Y 240.022,Z 1273.635,A -85,B 0,C 180,E1 11437.43,E2 11437.43} C_VEL
LIN {X 0,Y 240.006,Z 1274.591,A -85,B 0,C 180,E1 11433.115,E2 11433.115} C_VEL
LIN {X 0,Y 240.001,Z 1274.759,A -85,B 0,C 180,E1 11428.579,E2 11428.579} C_VEL
LIN {X 0,Y 240.006,Z 1274.065,A -85,B 0,C 180,E1 11424.033,E2 11424.033} C_VEL
LIN {X 0,Y 240.208,Z 1272.272,A -85,B 0,C 180,E1 11418.973,E2 11418.973} C_VEL
LIN {X 0,Y 241.068,Z 1269.431,A -85,B 0,C 180,E1 11413.877,E2 11413.877} C_VEL
LIN {X 0,Y 242.947,Z 1265.534,A -85,B 0,C 180,E1 11408.779,E2 11408.779} C_VEL
LIN {X 0,Y 246.058,Z 1260.558,A -85,B 0,C 180,E1 11403.722,E2 11403.722} C_VEL
LIN {X 0,Y 250.646,Z 1254.289,A -85,B 0,C 180,E1 11398.617,E2 11398.617} C_VEL
LIN {X 0,Y 257.68,Z 1245.793,A -85,B 0,C 180,E1 11393.041,E2 11393.041} C_VEL
LIN {X 0,Y 267.301,Z 1234.814,A -85,B 0,C 180,E1 11387.402,E2 11387.402} C_VEL
LIN {X 0,Y 276.756,Z 1224.352,A -85,B 0,C 180,E1 11383.066,E2 11383.066} C_VEL
LIN {X 0,Y 286.74,Z 1213.372,A -85,B 0,C 180,E1 11379.292,E2 11379.292} C_VEL
LIN {X 0,Y 298.543,Z 1200.236,A -85,B 0,C 180,E1 11375.545,E2 11375.545} C_VEL
LIN {X 0,Y 313.396,Z 1183.06,A -85,B 0,C 180,E1 11371.607,E2 11371.607} C_VEL
LIN {X 0,Y 325.756,Z 1168.048,A -85,B 0,C 180,E1 11368.81,E2 11368.81} C_VEL
LIN {X 0,Y 337.694,Z 1152.818,A -85,B 0,C 180,E1 11366.428,E2 11366.428} C_VEL
LIN {X 0,Y 350.575,Z 1135.421,A -85,B 0,C 180,E1 11364.147,E2 11364.147} C_VEL
LIN {X 0,Y 365.926,Z 1112.886,A -85,B 0,C 180,E1 11361.741,E2 11361.741} C_VEL
LIN {X 0,Y 377.436,Z 1094.437,A -85,B 0,C 180,E1 11360.124,E2 11360.124} C_VEL
LIN {X 0,Y 387.637,Z 1076.762,A -85,B 0,C 180,E1 11358.81,E2 11358.81} C_VEL
LIN {X 0,Y 397.529,Z 1058.066,A -85,B 0,C 180,E1 11357.615,E2 11357.615} C_VEL
LIN {X 0,Y 408.075,Z 1036.153,A -85,B 0,C 180,E1 11356.442,E2 11356.442} C_VEL
LIN {X 0,Y 418.791,Z 1010.652,A -85,B 0,C 180,E1 11355.332,E2 11355.332} C_VEL
LIN {X 0,Y 426.61,Z 989.277,A -85,B 0,C 180,E1 11354.573,E2 11354.573} C_VEL
LIN {X 0,Y 433.414,Z 967.937,A -85,B 0,C 180,E1 11353.949,E2 11353.949} C_VEL
LIN {X 0,Y 439.359,Z 946.102,A -85,B 0,C 180,E1 11353.43,E2 11353.43} C_VEL
LIN {X 0,Y 445.444,Z 918.446,A -85,B 0,C 180,E1 11352.905,E2 11352.905} C_VEL
LIN {X 0,Y 449.468,Z 892.248,A -85,B 0,C 180,E1 11352.48,E2 11352.48} C_VEL
LIN {X 0,Y 466.508,Z 727.691,A -85,B 0,C 180,E1 11350.116,E2 11350.116} C_VEL
LIN {X 0,Y 470.947,Z 684.945,A -85,B 0,C 180,E1 11349.502,E2 11349.502} C_VEL
LIN {X 0,Y 468.883,Z 680.982,A -85,B 0,C 180,E1 11347.474,E2 11347.474} C_VEL
LIN {X 0,Y 467.149,Z 677.377,A -85,B 0,C 180,E1 11345.158,E2 11345.158} C_VEL
LIN {X 0,Y 465.703,Z 673.691,A -85,B 0,C 180,E1 11341.353,E2 11341.353} C_VEL
LIN {X 0,Y 465.646,Z 673.101,A -85,B 0,C 180,E1 11340.615,E2 11340.615} C_VEL
LIN {X 0,Y 465.68,Z 673.248,A -85,B 0,C 180,E1 11338.524,E2 11338.524} C_VEL
LIN {X 0,Y 467.539,Z 678.162,A -85,B 0,C 180,E1 11333.738,E2 11333.738} C_VEL
LIN {X 0,Y 469.675,Z 682.498,A -85,B 0,C 180,E1 11331.183,E2 11331.183} C_VEL
LIN {X 0,Y 470.812,Z 684.933,A -85,B 0,C 180,E1 11330.089,E2 11330.089} C_VEL
LIN {X 0,Y 449.971,Z 885.374,A -85,B 0,C 180,E1 11327.225,E2 11327.225} C_VEL
LIN {X 0,Y 446.158,Z 910.297,A -85,B 0,C 180,E1 11326.823,E2 11326.823} C_VEL
LIN {X 0,Y 440.104,Z 938.583,A -85,B 0,C 180,E1 11326.241,E2 11326.241} C_VEL
LIN {X 0,Y 434.162,Z 960.733,A -85,B 0,C 180,E1 11325.659,E2 11325.659} C_VEL
LIN {X 0,Y 427.91,Z 980.623,A -85,B 0,C 180,E1 11325.028,E2 11325.028} C_VEL
LIN {X 0,Y 420.642,Z 1000.815,A -85,B 0,C 180,E1 11324.269,E2 11324.269} C_VEL
LIN {X 0,Y 411.043,Z 1024.272,A -85,B 0,C 180,E1 11323.217,E2 11323.217} C_VEL
LIN {X 0,Y 399.685,Z 1048.264,A -85,B 0,C 180,E1 11321.892,E2 11321.892} C_VEL
LIN {X 0,Y 389.446,Z 1067.602,A -85,B 0,C 180,E1 11320.626,E2 11320.626} C_VEL
LIN {X 0,Y 379.017,Z 1085.626,A -85,B 0,C 180,E1 11319.234,E2 11319.234} C_VEL
LIN {X 0,Y 367.657,Z 1103.707,A -85,B 0,C 180,E1 11317.592,E2 11317.592} C_VEL
LIN {X 0,Y 352.813,Z 1125.291,A -85,B 0,C 180,E1 11315.229,E2 11315.229} C_VEL
LIN {X 0,Y 340.077,Z 1142.238,A -85,B 0,C 180,E1 11312.96,E2 11312.96} C_VEL
LIN {X 0,Y 328.477,Z 1156.756,A -85,B 0,C 180,E1 11310.653,E2 11310.653} C_VEL
LIN {X 0,Y 316.869,Z 1170.528,A -85,B 0,C 180,E1 11308.064,E2 11308.064} C_VEL
LIN {X 0,Y 303.046,Z 1186.234,A -85,B 0,C 180,E1 11304.5,E2 11304.5} C_VEL
LIN {X 0,Y 289.5,Z 1200.695,A -85,B 0,C 180,E1 11300.354,E2 11300.354} C_VEL
LIN {X 0,Y 279.266,Z 1211.4,A -85,B 0,C 180,E1 11296.604,E2 11296.604} C_VEL
LIN {X 0,Y 269.94,Z 1221.071,A -85,B 0,C 180,E1 11292.513,E2 11292.513} C_VEL
LIN {X 0,Y 260.164,Z 1231.458,A -85,B 0,C 180,E1 11287.099,E2 11287.099} C_VEL
LIN {X 0,Y 252.27,Z 1240.015,A -85,B 0,C 180,E1 11281.266,E2 11281.266} C_VEL
LIN {X 0,Y 247.477,Z 1245.741,A -85,B 0,C 180,E1 11276.374,E2 11276.374} C_VEL
LIN {X 0,Y 244.025,Z 1250.399,A -85,B 0,C 180,E1 11271.375,E2 11271.375} C_VEL
LIN {X 0,Y 241.811,Z 1253.977,A -85,B 0,C 180,E1 11266.397,E2 11266.397} C_VEL
LIN {X 0,Y 240.621,Z 1256.546,A -85,B 0,C 180,E1 11261.494,E2 11261.494} C_VEL
LIN {X 0,Y 240.17,Z 1258.119,A -85,B 0,C 180,E1 11256.923,E2 11256.923} C_VEL
LIN {X 0,Y 240.03,Z 1258.896,A -85,B 0,C 180,E1 11252.615,E2 11252.615} C_VEL
LIN {X 0,Y 240.015,Z 1258.991,A -85,B 0,C 180,E1 11248.318,E2 11248.318} C_VEL
LIN {X 0,Y 240.128,Z 1258.34,A -85,B 0,C 180,E1 11243.774,E2 11243.774} C_VEL
LIN {X 0,Y 240.55,Z 1256.737,A -85,B 0,C 180,E1 11238.808,E2 11238.808} C_VEL
LIN {X 0,Y 241.697,Z 1254.24,A -85,B 0,C 180,E1 11233.898,E2 11233.898} C_VEL
LIN {X 0,Y 243.862,Z 1250.676,A -85,B 0,C 180,E1 11228.839,E2 11228.839} C_VEL
LIN {X 0,Y 247.23,Z 1246.082,A -85,B 0,C 180,E1 11223.833,E2 11223.833} C_VEL
LIN {X 0,Y 251.803,Z 1240.589,A -85,B 0,C 180,E1 11219.062,E2 11219.062} C_VEL
LIN {X 0,Y 258.072,Z 1233.649,A -85,B 0,C 180,E1 11214.184,E2 11214.184} C_VEL
LIN {X 0,Y 267.61,Z 1223.688,A -85,B 0,C 180,E1 11208.588,E2 11208.588} C_VEL
LIN {X 0,Y 278.205,Z 1212.581,A -85,B 0,C 180,E1 11203.736,E2 11203.736} C_VEL
LIN {X 0,Y 288.322,Z 1202.011,A -85,B 0,C 180,E1 11199.956,E2 11199.956} C_VEL
LIN {X 0,Y 299.254,Z 1190.36,A -85,B 0,C 180,E1 11196.495,E2 11196.495} C_VEL
LIN {X 0,Y 312.945,Z 1175.319,A -85,B 0,C 180,E1 11192.817,E2 11192.817} C_VEL
LIN {X 0,Y 326.74,Z 1159.047,A -85,B 0,C 180,E1 11189.636,E2 11189.636} C_VEL
LIN {X 0,Y 338.586,Z 1144.328,A -85,B 0,C 180,E1 11187.241,E2 11187.241} C_VEL
LIN {X 0,Y 350.154,Z 1129.066,A -85,B 0,C 180,E1 11185.137,E2 11185.137} C_VEL
LIN {X 0,Y 362.561,Z 1111.57,A -85,B 0,C 180,E1 11183.101,E2 11183.101} C_VEL
LIN {X 0,Y 377.421,Z 1088.579,A -85,B 0,C 180,E1 11180.908,E2 11180.908} C_VEL
LIN {X 0,Y 388.567,Z 1069.512,A -85,B 0,C 180,E1 11179.409,E2 11179.409} C_VEL
LIN {X 0,Y 398.38,Z 1051.168,A -85,B 0,C 180,E1 11178.186,E2 11178.186} C_VEL
LIN {X 0,Y 407.498,Z 1032.376,A -85,B 0,C 180,E1 11177.102,E2 11177.102} C_VEL
LIN {X 0,Y 418.044,Z 1008.175,A -85,B 0,C 180,E1 11175.936,E2 11175.936} C_VEL
LIN {X 0,Y 427.003,Z 983.913,A -85,B 0,C 180,E1 11174.988,E2 11174.988} C_VEL
LIN {X 0,Y 433.684,Z 963.044,A -85,B 0,C 180,E1 11174.312,E2 11174.312} C_VEL
LIN {X 0,Y 439.513,Z 941.714,A -85,B 0,C 180,E1 11173.737,E2 11173.737} C_VEL
LIN {X 0,Y 444.599,Z 919.281,A -85,B 0,C 180,E1 11173.247,E2 11173.247} C_VEL
LIN {X 0,Y 449.562,Z 890.361,A -85,B 0,C 180,E1 11172.753,E2 11172.753} C_VEL
LIN {X 0,Y 449.859,Z 887.957,A -85,B 0,C 180,E1 11172.717,E2 11172.717} C_VEL
LIN {X 0,Y 450.568,Z 880.453,A -85,B 0,C 180,E1 11172.477,E2 11172.477} C_VEL
LIN {X 0,Y 451.438,Z 860.938,A -85,B 0,C 180,E1 11171.416,E2 11171.416} C_VEL
LIN {X 0,Y 451.947,Z 854.465,A -85,B 0,C 180,E1 11171.23,E2 11171.23} C_VEL
LIN {X 0,Y 469.07,Z 691.205,A -85,B 0,C 180,E1 11168.921,E2 11168.921} C_VEL
LIN {X 0,Y 467.761,Z 688.524,A -85,B 0,C 180,E1 11167.492,E2 11167.492} C_VEL
LIN {X 0,Y 466.303,Z 685.319,A -85,B 0,C 180,E1 11165.414,E2 11165.414} C_VEL
LIN {X 0,Y 464.922,Z 681.061,A -85,B 0,C 180,E1 11160.739,E2 11160.739} C_VEL
LIN {X 0,Y 464.942,Z 681.402,A -85,B 0,C 180,E1 11159.137,E2 11159.137} C_VEL
LIN {X 0,Y 466.67,Z 686.147,A -85,B 0,C 180,E1 11154.405,E2 11154.405} C_VEL
LIN {X 0,Y 468.791,Z 690.588,A -85,B 0,C 180,E1 11151.784,E2 11151.784} C_VEL
LIN {X 0,Y 469.178,Z 691.657,A -85,B 0,C 180,E1 11151.366,E2 11151.366} C_VEL
LIN {X 0,Y 448.037,Z 891.732,A -85,B 0,C 180,E1 11148.536,E2 11148.536} C_VEL
LIN {X 0,Y 444.063,Z 917.339,A -85,B 0,C 180,E1 11148.129,E2 11148.129} C_VEL
LIN {X 0,Y 437.851,Z 945.479,A -85,B 0,C 180,E1 11147.611,E2 11147.611} C_VEL
LIN {X 0,Y 431.858,Z 967.271,A -85,B 0,C 180,E1 11147.11,E2 11147.11} C_VEL
LIN {X 0,Y 425.182,Z 988.01,A -85,B 0,C 180,E1 11146.524,E2 11146.524} C_VEL
LIN {X 0,Y 417.247,Z 1009.493,A -85,B 0,C 180,E1 11145.788,E2 11145.788} C_VEL
LIN {X 0,Y 406.367,Z 1035.166,A -85,B 0,C 180,E1 11144.708,E2 11144.708} C_VEL
LIN {X 0,Y 395.506,Z 1057.414,A -85,B 0,C 180,E1 11143.552,E2 11143.552} C_VEL
LIN {X 0,Y 385.515,Z 1076.005,A -85,B 0,C 180,E1 11142.395,E2 11142.395} C_VEL
LIN {X 0,Y 375.172,Z 1093.625,A -85,B 0,C 180,E1 11141.119,E2 11141.119} C_VEL
LIN {X 0,Y 363.576,Z 1111.878,A -85,B 0,C 180,E1 11139.557,E2 11139.557} C_VEL
LIN {X 0,Y 348.48,Z 1133.708,A -85,B 0,C 180,E1 11137.295,E2 11137.295} C_VEL
LIN {X 0,Y 334.507,Z 1152.145,A -85,B 0,C 180,E1 11134.93,E2 11134.93} C_VEL
LIN {X 0,Y 322.21,Z 1167.43,A -85,B 0,C 180,E1 11132.575,E2 11132.575} C_VEL
LIN {X 0,Y 309.813,Z 1182.053,A -85,B 0,C 180,E1 11129.887,E2 11129.887} C_VEL
LIN {X 0,Y 295.012,Z 1198.698,A -85,B 0,C 180,E1 11126.149,E2 11126.149} C_VEL
LIN {X 0,Y 282.073,Z 1212.533,A -85,B 0,C 180,E1 11122.242,E2 11122.242} C_VEL
LIN {X 0,Y 271.461,Z 1223.706,A -85,B 0,C 180,E1 11118.404,E2 11118.404} C_VEL
LIN {X 0,Y 262.066,Z 1233.611,A -85,B 0,C 180,E1 11114.295,E2 11114.295} C_VEL
LIN {X 0,Y 252.086,Z 1244.403,A -85,B 0,C 180,E1 11108.818,E2 11108.818} C_VEL
LIN {X 0,Y 243.934,Z 1253.582,A -85,B 0,C 180,E1 11102.767,E2 11102.767} C_VEL
LIN {X 0,Y 238.822,Z 1260.031,A -85,B 0,C 180,E1 11097.427,E2 11097.427} C_VEL
LIN {X 0,Y 235.366,Z 1265.103,A -85,B 0,C 180,E1 11092.163,E2 11092.163} C_VEL
LIN {X 0,Y 233.336,Z 1268.878,A -85,B 0,C 180,E1 11087.137,E2 11087.137} C_VEL
LIN {X 0,Y 232.339,Z 1271.65,A -85,B 0,C 180,E1 11082.184,E2 11082.184} C_VEL
LIN {X 0,Y 232.029,Z 1273.515,A -85,B 0,C 180,E1 11077.19,E2 11077.19} C_VEL
LIN {X 0,Y 232.01,Z 1274.353,A -85,B 0,C 180,E1 11072.976,E2 11072.976} C_VEL
LIN {X 0,Y 232.007,Z 1274.496,A -85,B 0,C 180,E1 11068.53,E2 11068.53} C_VEL
LIN {X 0,Y 232.012,Z 1273.801,A -85,B 0,C 180,E1 11063.827,E2 11063.827} C_VEL
LIN {X 0,Y 232.251,Z 1272.006,A -85,B 0,C 180,E1 11058.59,E2 11058.59} C_VEL
LIN {X 0,Y 233.202,Z 1269.162,A -85,B 0,C 180,E1 11053.318,E2 11053.318} C_VEL
LIN {X 0,Y 235.253,Z 1265.261,A -85,B 0,C 180,E1 11048.049,E2 11048.049} C_VEL
LIN {X 0,Y 238.613,Z 1260.284,A -85,B 0,C 180,E1 11042.836,E2 11042.836} C_VEL
LIN {X 0,Y 243.372,Z 1254.199,A -85,B 0,C 180,E1 11037.732,E2 11037.732} C_VEL
LIN {X 0,Y 250.308,Z 1246.244,A -85,B 0,C 180,E1 11032.341,E2 11032.341} C_VEL
LIN {X 0,Y 261.149,Z 1234.536,A -85,B 0,C 180,E1 11026.148,E2 11026.148} C_VEL
LIN {X 0,Y 270.911,Z 1224.215,A -85,B 0,C 180,E1 11021.812,E2 11021.812} C_VEL
LIN {X 0,Y 280.904,Z 1213.679,A -85,B 0,C 180,E1 11018.145,E2 11018.145} C_VEL
LIN {X 0,Y 292.494,Z 1201.252,A -85,B 0,C 180,E1 11014.548,E2 11014.548} C_VEL
LIN {X 0,Y 307.094,Z 1185.109,A -85,B 0,C 180,E1 11010.743,E2 11010.743} C_VEL
LIN {X 0,Y 321.424,Z 1168.224,A -85,B 0,C 180,E1 11007.577,E2 11007.577} C_VEL
LIN {X 0,Y 333.685,Z 1153.009,A -85,B 0,C 180,E1 11005.21,E2 11005.21} C_VEL
LIN {X 0,Y 346.094,Z 1136.683,A -85,B 0,C 180,E1 11003.076,E2 11003.076} C_VEL
LIN {X 0,Y 360.946,Z 1115.684,A -85,B 0,C 180,E1 11000.811,E2 11000.811} C_VEL
LIN {X 0,Y 374.262,Z 1094.835,A -85,B 0,C 180,E1 10998.989,E2 10998.989} C_VEL
LIN {X 0,Y 385.026,Z 1076.55,A -85,B 0,C 180,E1 10997.655,E2 10997.655} C_VEL
LIN {X 0,Y 395.124,Z 1057.791,A -85,B 0,C 180,E1 10996.481,E2 10996.481} C_VEL
LIN {X 0,Y 406.272,Z 1034.973,A -85,B 0,C 180,E1 10995.292,E2 10995.292} C_VEL
LIN {X 0,Y 417.151,Z 1009.241,A -85,B 0,C 180,E1 10994.211,E2 10994.211} C_VEL
LIN {X 0,Y 424.937,Z 988.144,A -85,B 0,C 180,E1 10993.488,E2 10993.488} C_VEL
LIN {X 0,Y 431.761,Z 966.92,A -85,B 0,C 180,E1 10992.889,E2 10992.889} C_VEL
LIN {X 0,Y 437.978,Z 944.201,A -85,B 0,C 180,E1 10992.369,E2 10992.369} C_VEL
LIN {X 0,Y 444.379,Z 914.246,A -85,B 0,C 180,E1 10991.827,E2 10991.827} C_VEL
LIN {X 0,Y 447.935,Z 890.853,A -85,B 0,C 180,E1 10991.457,E2 10991.457} C_VEL
LIN {X 0,Y 468.985,Z 691.315,A -85,B 0,C 180,E1 10988.633,E2 10988.633} C_VEL
LIN {X 0,Y 467.572,Z 688.509,A -85,B 0,C 180,E1 10987.125,E2 10987.125} C_VEL
LIN {X 0,Y 466.092,Z 685.257,A -85,B 0,C 180,E1 10985.046,E2 10985.046} C_VEL
LIN {X 0,Y 464.702,Z 681.418,A -85,B 0,C 180,E1 10981.11,E2 10981.11} C_VEL
LIN {X 0,Y 464.644,Z 681.049,A -85,B 0,C 180,E1 10980.37,E2 10980.37} C_VEL
LIN {X 0,Y 464.694,Z 681.281,A -85,B 0,C 180,E1 10978.52,E2 10978.52} C_VEL
LIN {X 0,Y 466.432,Z 685.966,A -85,B 0,C 180,E1 10973.909,E2 10973.909} C_VEL
LIN {X 0,Y 468.504,Z 690.321,A -85,B 0,C 180,E1 10971.346,E2 10971.346} C_VEL
LIN {X 0,Y 468.85,Z 691.313,A -85,B 0,C 180,E1 10970.966,E2 10970.966} C_VEL
LIN {X 0,Y 448.255,Z 885.766,A -85,B 0,C 180,E1 10968.222,E2 10968.222} C_VEL
LIN {X 0,Y 444.319,Z 911.063,A -85,B 0,C 180,E1 10967.82,E2 10967.82} C_VEL
LIN {X 0,Y 438.211,Z 939.073,A -85,B 0,C 180,E1 10967.254,E2 10967.254} C_VEL
LIN {X 0,Y 432.242,Z 961.007,A -85,B 0,C 180,E1 10966.691,E2 10966.691} C_VEL
LIN {X 0,Y 425.901,Z 980.896,A -85,B 0,C 180,E1 10966.075,E2 10966.075} C_VEL
LIN {X 0,Y 418.504,Z 1001.145,A -85,B 0,C 180,E1 10965.33,E2 10965.33} C_VEL
LIN {X 0,Y 408.653,Z 1024.839,A -85,B 0,C 180,E1 10964.29,E2 10964.29} C_VEL
LIN {X 0,Y 397.234,Z 1048.536,A -85,B 0,C 180,E1 10963.006,E2 10963.006} C_VEL
LIN {X 0,Y 386.936,Z 1067.667,A -85,B 0,C 180,E1 10961.779,E2 10961.779} C_VEL
LIN {X 0,Y 376.199,Z 1085.899,A -85,B 0,C 180,E1 10960.397,E2 10960.397} C_VEL
LIN {X 0,Y 365.181,Z 1103.11,A -85,B 0,C 180,E1 10958.866,E2 10958.866} C_VEL
LIN {X 0,Y 351.397,Z 1123.002,A -85,B 0,C 180,E1 10956.766,E2 10956.766} C_VEL
LIN {X 0,Y 337.071,Z 1141.676,A -85,B 0,C 180,E1 10954.336,E2 10954.336} C_VEL
LIN {X 0,Y 324.9,Z 1156.547,A -85,B 0,C 180,E1 10952.014,E2 10952.014} C_VEL
LIN {X 0,Y 313.101,Z 1170.178,A -85,B 0,C 180,E1 10949.485,E2 10949.485} C_VEL
LIN {X 0,Y 300.264,Z 1184.309,A -85,B 0,C 180,E1 10946.337,E2 10946.337} C_VEL
LIN {X 0,Y 285.383,Z 1199.848,A -85,B 0,C 180,E1 10942.01,E2 10942.01} C_VEL
LIN {X 0,Y 274.112,Z 1211.172,A -85,B 0,C 180,E1 10938.067,E2 10938.067} C_VEL
LIN {X 0,Y 264.528,Z 1220.671,A -85,B 0,C 180,E1 10934.05,E2 10934.05} C_VEL
LIN {X 0,Y 255.432,Z 1229.773,A -85,B 0,C 180,E1 10929.341,E2 10929.341} C_VEL
LIN {X 0,Y 245.789,Z 1239.701,A -85,B 0,C 180,E1 10922.741,E2 10922.741} C_VEL
LIN {X 0,Y 240.326,Z 1245.768,A -85,B 0,C 180,E1 10917.491,E2 10917.491} C_VEL
LIN {X 0,Y 236.409,Z 1250.638,A -85,B 0,C 180,E1 10912.14,E2 10912.14} C_VEL
LIN {X 0,Y 234.045,Z 1254.142,A -85,B 0,C 180,E1 10907.132,E2 10907.132} C_VEL
LIN {X 0,Y 232.749,Z 1256.704,A -85,B 0,C 180,E1 10902.14,E2 10902.14} C_VEL
LIN {X 0,Y 232.201,Z 1258.319,A -85,B 0,C 180,E1 10897.411,E2 10897.411} C_VEL
LIN {X 0,Y 232.038,Z 1259.137,A -85,B 0,C 180,E1 10892.953,E2 10892.953} C_VEL
LIN {X 0,Y 232.012,Z 1259.275,A -85,B 0,C 180,E1 10888.507,E2 10888.507} C_VEL
LIN {X 0,Y 232.145,Z 1258.604,A -85,B 0,C 180,E1 10883.559,E2 10883.559} C_VEL
LIN {X 0,Y 232.638,Z 1256.965,A -85,B 0,C 180,E1 10878.335,E2 10878.335} C_VEL
LIN {X 0,Y 233.941,Z 1254.355,A -85,B 0,C 180,E1 10873.093,E2 10873.093} C_VEL
LIN {X 0,Y 236.357,Z 1250.746,A -85,B 0,C 180,E1 10867.872,E2 10867.872} C_VEL
LIN {X 0,Y 240.062,Z 1246.107,A -85,B 0,C 180,E1 10862.721,E2 10862.721} C_VEL
LIN {X 0,Y 245.439,Z 1240.107,A -85,B 0,C 180,E1 10857.459,E2 10857.459} C_VEL
LIN {X 0,Y 253.87,Z 1231.497,A -85,B 0,C 180,E1 10851.505,E2 10851.505} C_VEL
LIN {X 0,Y 263.993,Z 1221.276,A -85,B 0,C 180,E1 10846.112,E2 10846.112} C_VEL
LIN {X 0,Y 273.512,Z 1211.847,A -85,B 0,C 180,E1 10842.077,E2 10842.077} C_VEL
LIN {X 0,Y 283.601,Z 1201.722,A -85,B 0,C 180,E1 10838.481,E2 10838.481} C_VEL
LIN {X 0,Y 295.47,Z 1189.506,A -85,B 0,C 180,E1 10834.884,E2 10834.884} C_VEL
LIN {X 0,Y 311.139,Z 1172.572,A -85,B 0,C 180,E1 10830.892,E2 10830.892} C_VEL
LIN {X 0,Y 323.415,Z 1158.484,A -85,B 0,C 180,E1 10828.211,E2 10828.211} C_VEL
LIN {X 0,Y 334.857,Z 1144.631,A -85,B 0,C 180,E1 10825.989,E2 10825.989} C_VEL
LIN {X 0,Y 346.357,Z 1129.834,A -85,B 0,C 180,E1 10823.968,E2 10823.968} C_VEL
LIN {X 0,Y 358.634,Z 1112.933,A -85,B 0,C 180,E1 10822.013,E2 10822.013} C_VEL
LIN {X 0,Y 373.307,Z 1090.937,A -85,B 0,C 180,E1 10819.913,E2 10819.913} C_VEL
LIN {X 0,Y 385.522,Z 1070.504,A -85,B 0,C 180,E1 10818.319,E2 10818.319} C_VEL
LIN {X 0,Y 395.5,Z 1052.234,A -85,B 0,C 180,E1 10817.117,E2 10817.117} C_VEL
LIN {X 0,Y 404.764,Z 1033.529,A -85,B 0,C 180,E1 10816.053,E2 10816.053} C_VEL
LIN {X 0,Y 414.169,Z 1012.432,A -85,B 0,C 180,E1 10815.042,E2 10815.042} C_VEL
LIN {X 0,Y 424.557,Z 985.447,A -85,B 0,C 180,E1 10813.983,E2 10813.983} C_VEL
LIN {X 0,Y 431.547,Z 964.035,A -85,B 0,C 180,E1 10813.299,E2 10813.299} C_VEL
LIN {X 0,Y 437.539,Z 942.506,A -85,B 0,C 180,E1 10812.729,E2 10812.729} C_VEL
LIN {X 0,Y 442.594,Z 920.636,A -85,B 0,C 180,E1 10812.259,E2 10812.259} C_VEL
LIN {X 0,Y 447.541,Z 893.166,A -85,B 0,C 180,E1 10811.792,E2 10811.792} C_VEL
LIN {X 0,Y 451.947,Z 854.465,A -85,B 0,C 180,E1 10811.23,E2 10811.23} C_VEL
LIN {X 0,Y 452.535,Z 846.938,A -85,B 0,C 180,E1 10810.997,E2 10810.997} C_VEL
LIN {X 0,Y 453.458,Z 827.418,A -85,B 0,C 180,E1 10809.94,E2 10809.94} C_VEL
LIN {X 0,Y 454.022,Z 820.94,A -85,B 0,C 180,E1 10809.76,E2 10809.76} C_VEL
LIN {X 0,Y 467.235,Z 697.468,A -85,B 0,C 180,E1 10808.03,E2 10808.03} C_VEL
LIN {X 0,Y 465.25,Z 693.201,A -85,B 0,C 180,E1 10805.303,E2 10805.303} C_VEL
LIN {X 0,Y 463.939,Z 689.006,A -85,B 0,C 180,E1 10800.617,E2 10800.617} C_VEL
LIN {X 0,Y 463.957,Z 689.281,A -85,B 0,C 180,E1 10799.259,E2 10799.259} C_VEL
LIN {X 0,Y 465.567,Z 693.949,A -85,B 0,C 180,E1 10794.578,E2 10794.578} C_VEL
LIN {X 0,Y 467.336,Z 697.873,A -85,B 0,C 180,E1 10792.253,E2 10792.253} C_VEL
LIN {X 0,Y 446.51,Z 891.461,A -85,B 0,C 180,E1 10789.549,E2 10789.549} C_VEL
LIN {X 0,Y 442.477,Z 917.091,A -85,B 0,C 180,E1 10789.149,E2 10789.149} C_VEL
LIN {X 0,Y 436.192,Z 945.229,A -85,B 0,C 180,E1 10788.645,E2 10788.645} C_VEL
LIN {X 0,Y 430.128,Z 967.015,A -85,B 0,C 180,E1 10788.158,E2 10788.158} C_VEL
LIN {X 0,Y 423.349,Z 987.805,A -85,B 0,C 180,E1 10787.589,E2 10787.589} C_VEL
LIN {X 0,Y 415.325,Z 1009.233,A -85,B 0,C 180,E1 10786.876,E2 10786.876} C_VEL
LIN {X 0,Y 404.291,Z 1034.903,A -85,B 0,C 180,E1 10785.824,E2 10785.824} C_VEL
LIN {X 0,Y 393.402,Z 1056.887,A -85,B 0,C 180,E1 10784.712,E2 10784.712} C_VEL
LIN {X 0,Y 383.127,Z 1075.703,A -85,B 0,C 180,E1 10783.571,E2 10783.571} C_VEL
LIN {X 0,Y 372.163,Z 1094.032,A -85,B 0,C 180,E1 10782.27,E2 10782.27} C_VEL
LIN {X 0,Y 358.98,Z 1114.302,A -85,B 0,C 180,E1 10780.547,E2 10780.547} C_VEL
LIN {X 0,Y 343.39,Z 1135.986,A -85,B 0,C 180,E1 10778.271,E2 10778.271} C_VEL
LIN {X 0,Y 330.673,Z 1152.342,A -85,B 0,C 180,E1 10776.175,E2 10776.175} C_VEL
LIN {X 0,Y 318.434,Z 1167.158,A -85,B 0,C 180,E1 10773.914,E2 10773.914} C_VEL
LIN {X 0,Y 305.747,Z 1181.702,A -85,B 0,C 180,E1 10771.266,E2 10771.266} C_VEL
LIN {X 0,Y 290.259,Z 1198.565,A -85,B 0,C 180,E1 10767.494,E2 10767.494} C_VEL
LIN {X 0,Y 276.979,Z 1212.257,A -85,B 0,C 180,E1 10763.624,E2 10763.624} C_VEL
LIN {X 0,Y 265.921,Z 1223.43,A -85,B 0,C 180,E1 10759.767,E2 10759.767} C_VEL
LIN {X 0,Y 256.077,Z 1233.335,A -85,B 0,C 180,E1 10755.618,E2 10755.618} C_VEL
LIN {X 0,Y 245.575,Z 1244.128,A -85,B 0,C 180,E1 10750.051,E2 10750.051} C_VEL
LIN {X 0,Y 236.921,Z 1253.308,A -85,B 0,C 180,E1 10743.866,E2 10743.866} C_VEL
LIN {X 0,Y 231.445,Z 1259.753,A -85,B 0,C 180,E1 10738.385,E2 10738.385} C_VEL
LIN {X 0,Y 227.761,Z 1264.78,A -85,B 0,C 180,E1 10733.01,E2 10733.01} C_VEL
LIN {X 0,Y 225.535,Z 1268.562,A -85,B 0,C 180,E1 10727.824,E2 10727.824} C_VEL
LIN {X 0,Y 224.39,Z 1271.389,A -85,B 0,C 180,E1 10722.611,E2 10722.611} C_VEL
LIN {X 0,Y 224.025,Z 1273.178,A -85,B 0,C 180,E1 10717.706,E2 10717.706} C_VEL
LIN {X 0,Y 224.012,Z 1274.066,A -85,B 0,C 180,E1 10713.338,E2 10713.338} C_VEL
LIN {X 0,Y 224.003,Z 1274.257,A -85,B 0,C 180,E1 10708.733,E2 10708.733} C_VEL
LIN {X 0,Y 224.014,Z 1273.608,A -85,B 0,C 180,E1 10703.863,E2 10703.863} C_VEL
LIN {X 0,Y 224.295,Z 1271.739,A -85,B 0,C 180,E1 10698.179,E2 10698.179} C_VEL
LIN {X 0,Y 225.358,Z 1268.892,A -85,B 0,C 180,E1 10692.719,E2 10692.719} C_VEL
LIN {X 0,Y 227.603,Z 1264.99,A -85,B 0,C 180,E1 10687.271,E2 10687.271} C_VEL
LIN {X 0,Y 231.219,Z 1260.009,A -85,B 0,C 180,E1 10681.892,E2 10681.892} C_VEL
LIN {X 0,Y 236.324,Z 1253.923,A -85,B 0,C 180,E1 10676.646,E2 10676.646} C_VEL
LIN {X 0,Y 244.049,Z 1245.602,A -85,B 0,C 180,E1 10670.896,E2 10670.896} C_VEL
LIN {X 0,Y 255.119,Z 1234.256,A -85,B 0,C 180,E1 10664.832,E2 10664.832} C_VEL
LIN {X 0,Y 265.344,Z 1223.935,A -85,B 0,C 180,E1 10660.45,E2 10660.45} C_VEL
LIN {X 0,Y 275.852,Z 1213.306,A -85,B 0,C 180,E1 10656.733,E2 10656.733} C_VEL
LIN {X 0,Y 287.789,Z 1200.973,A -85,B 0,C 180,E1 10653.163,E2 10653.163} C_VEL
LIN {X 0,Y 302.861,Z 1184.853,A -85,B 0,C 180,E1 10649.38,E2 10649.38} C_VEL
LIN {X 0,Y 316.903,Z 1168.804,A -85,B 0,C 180,E1 10646.379,E2 10646.379} C_VEL
LIN {X 0,Y 329.453,Z 1153.67,A -85,B 0,C 180,E1 10644.029,E2 10644.029} C_VEL
LIN {X 0,Y 341.736,Z 1137.946,A -85,B 0,C 180,E1 10641.978,E2 10641.978} C_VEL
LIN {X 0,Y 354.774,Z 1120.101,A -85,B 0,C 180,E1 10640.032,E2 10640.032} C_VEL
LIN {X 0,Y 369.995,Z 1097.257,A -85,B 0,C 180,E1 10637.996,E2 10637.996} C_VEL
LIN {X 0,Y 381.762,Z 1077.757,A -85,B 0,C 180,E1 10636.578,E2 10636.578} C_VEL
LIN {X 0,Y 392.013,Z 1059.152,A -85,B 0,C 180,E1 10635.426,E2 10635.426} C_VEL
LIN {X 0,Y 401.815,Z 1039.616,A -85,B 0,C 180,E1 10634.409,E2 10634.409} C_VEL
LIN {X 0,Y 412.573,Z 1015.688,A -85,B 0,C 180,E1 10633.373,E2 10633.373} C_VEL
LIN {X 0,Y 422.373,Z 990.02,A -85,B 0,C 180,E1 10632.486,E2 10632.486} C_VEL
LIN {X 0,Y 429.352,Z 968.873,A -85,B 0,C 180,E1 10631.895,E2 10631.895} C_VEL
LIN {X 0,Y 435.303,Z 947.815,A -85,B 0,C 180,E1 10631.414,E2 10631.414} C_VEL
LIN {X 0,Y 440.685,Z 924.845,A -85,B 0,C 180,E1 10630.988,E2 10630.988} C_VEL
LIN {X 0,Y 445.937,Z 894.256,A -85,B 0,C 180,E1 10630.498,E2 10630.498} C_VEL
LIN {X 0,Y 452.798,Z 831.832,A -85,B 0,C 180,E1 10629.612,E2 10629.612} C_VEL
LIN {X 0,Y 467.119,Z 697.557,A -85,B 0,C 180,E1 10627.732,E2 10627.732} C_VEL
LIN {X 0,Y 464.96,Z 693.036,A -85,B 0,C 180,E1 10624.811,E2 10624.811} C_VEL
LIN {X 0,Y 463.712,Z 689.298,A -85,B 0,C 180,E1 10620.988,E2 10620.988} C_VEL
LIN {X 0,Y 463.642,Z 688.983,A -85,B 0,C 180,E1 10619.753,E2 10619.753} C_VEL
LIN {X 0,Y 463.707,Z 689.162,A -85,B 0,C 180,E1 10618.641,E2 10618.641} C_VEL
LIN {X 0,Y 465.365,Z 693.878,A -85,B 0,C 180,E1 10614.018,E2 10614.018} C_VEL
LIN {X 0,Y 467.023,Z 697.47,A -85,B 0,C 180,E1 10611.855,E2 10611.855} C_VEL
LIN {X 0,Y 446.69,Z 886.051,A -85,B 0,C 180,E1 10609.227,E2 10609.227} C_VEL
LIN {X 0,Y 442.671,Z 911.504,A -85,B 0,C 180,E1 10608.831,E2 10608.831} C_VEL
LIN {X 0,Y 436.512,Z 939.347,A -85,B 0,C 180,E1 10608.281,E2 10608.281} C_VEL
LIN {X 0,Y 430.463,Z 961.28,A -85,B 0,C 180,E1 10607.732,E2 10607.732} C_VEL
LIN {X 0,Y 424.035,Z 981.168,A -85,B 0,C 180,E1 10607.131,E2 10607.131} C_VEL
LIN {X 0,Y 416.386,Z 1001.797,A -85,B 0,C 180,E1 10606.389,E2 10606.389} C_VEL
LIN {X 0,Y 406.106,Z 1026.106,A -85,B 0,C 180,E1 10605.342,E2 10605.342} C_VEL
LIN {X 0,Y 394.552,Z 1049.532,A -85,B 0,C 180,E1 10604.091,E2 10604.091} C_VEL
LIN {X 0,Y 384.154,Z 1068.482,A -85,B 0,C 180,E1 10602.895,E2 10602.895} C_VEL
LIN {X 0,Y 373.126,Z 1086.832,A -85,B 0,C 180,E1 10601.524,E2 10601.524} C_VEL
LIN {X 0,Y 360.921,Z 1105.456,A -85,B 0,C 180,E1 10599.88,E2 10599.88} C_VEL
LIN {X 0,Y 345.108,Z 1127.29,A -85,B 0,C 180,E1 10597.527,E2 10597.527} C_VEL
LIN {X 0,Y 332.889,Z 1142.786,A -85,B 0,C 180,E1 10595.495,E2 10595.495} C_VEL
LIN {X 0,Y 321.093,Z 1156.822,A -85,B 0,C 180,E1 10593.32,E2 10593.32} C_VEL
LIN {X 0,Y 309.086,Z 1170.321,A -85,B 0,C 180,E1 10590.838,E2 10590.838} C_VEL
LIN {X 0,Y 295.955,Z 1184.344,A -85,B 0,C 180,E1 10587.737,E2 10587.737} C_VEL
LIN {X 0,Y 280.324,Z 1200.124,A -85,B 0,C 180,E1 10583.355,E2 10583.355} C_VEL
LIN {X 0,Y 268.606,Z 1211.448,A -85,B 0,C 180,E1 10579.392,E2 10579.392} C_VEL
LIN {X 0,Y 258.603,Z 1220.946,A -85,B 0,C 180,E1 10575.334,E2 10575.334} C_VEL
LIN {X 0,Y 249.036,Z 1230.049,A -85,B 0,C 180,E1 10570.558,E2 10570.558} C_VEL
LIN {X 0,Y 238.85,Z 1239.975,A -85,B 0,C 180,E1 10563.818,E2 10563.818} C_VEL
LIN {X 0,Y 232.975,Z 1246.091,A -85,B 0,C 180,E1 10558.378,E2 10558.378} C_VEL
LIN {X 0,Y 228.786,Z 1250.94,A -85,B 0,C 180,E1 10552.876,E2 10552.876} C_VEL
LIN {X 0,Y 226.251,Z 1254.41,A -85,B 0,C 180,E1 10547.741,E2 10547.741} C_VEL
LIN {X 0,Y 224.832,Z 1256.97,A -85,B 0,C 180,E1 10542.574,E2 10542.574} C_VEL
LIN {X 0,Y 224.207,Z 1258.648,A -85,B 0,C 180,E1 10537.419,E2 10537.419} C_VEL
LIN {X 0,Y 224.04,Z 1259.421,A -85,B 0,C 180,E1 10532.802,E2 10532.802} C_VEL
LIN {X 0,Y 224.026,Z 1259.516,A -85,B 0,C 180,E1 10528.198,E2 10528.198} C_VEL
LIN {X 0,Y 224.164,Z 1258.867,A -85,B 0,C 180,E1 10523.329,E2 10523.329} C_VEL
LIN {X 0,Y 224.719,Z 1257.23,A -85,B 0,C 180,E1 10517.918,E2 10517.918} C_VEL
LIN {X 0,Y 226.044,Z 1254.775,A -85,B 0,C 180,E1 10512.749,E2 10512.749} C_VEL
LIN {X 0,Y 228.603,Z 1251.214,A -85,B 0,C 180,E1 10507.351,E2 10507.351} C_VEL
LIN {X 0,Y 232.524,Z 1246.622,A -85,B 0,C 180,E1 10502.038,E2 10502.038} C_VEL
LIN {X 0,Y 238.11,Z 1240.742,A -85,B 0,C 180,E1 10496.685,E2 10496.685} C_VEL
LIN {X 0,Y 246.249,Z 1232.822,A -85,B 0,C 180,E1 10490.985,E2 10490.985} C_VEL
LIN {X 0,Y 257.117,Z 1222.444,A -85,B 0,C 180,E1 10485.25,E2 10485.25} C_VEL
LIN {X 0,Y 267.467,Z 1212.622,A -85,B 0,C 180,E1 10480.951,E2 10480.951} C_VEL
LIN {X 0,Y 277.911,Z 1202.555,A -85,B 0,C 180,E1 10477.321,E2 10477.321} C_VEL
LIN {X 0,Y 289.296,Z 1191.257,A -85,B 0,C 180,E1 10473.941,E2 10473.941} C_VEL
LIN {X 0,Y 303.579,Z 1176.552,A -85,B 0,C 180,E1 10470.34,E2 10470.34} C_VEL
LIN {X 0,Y 318.862,Z 1159.586,A -85,B 0,C 180,E1 10467.044,E2 10467.044} C_VEL
LIN {X 0,Y 331.317,Z 1144.899,A -85,B 0,C 180,E1 10464.704,E2 10464.704} C_VEL
LIN {X 0,Y 343.094,Z 1130.101,A -85,B 0,C 180,E1 10462.711,E2 10462.711} C_VEL
LIN {X 0,Y 355.239,Z 1113.747,A -85,B 0,C 180,E1 10460.844,E2 10460.844} C_VEL
LIN {X 0,Y 369.784,Z 1092.523,A -85,B 0,C 180,E1 10458.833,E2 10458.833} C_VEL
LIN {X 0,Y 383.036,Z 1070.767,A -85,B 0,C 180,E1 10457.161,E2 10457.161} C_VEL
LIN {X 0,Y 393.184,Z 1052.496,A -85,B 0,C 180,E1 10455.985,E2 10455.985} C_VEL
LIN {X 0,Y 402.598,Z 1033.789,A -85,B 0,C 180,E1 10454.945,E2 10454.945} C_VEL
LIN {X 0,Y 412.145,Z 1012.691,A -85,B 0,C 180,E1 10453.957,E2 10453.957} C_VEL
LIN {X 0,Y 422.682,Z 985.703,A -85,B 0,C 180,E1 10452.923,E2 10452.923} C_VEL
LIN {X 0,Y 430.019,Z 963.458,A -85,B 0,C 180,E1 10452.232,E2 10452.232} C_VEL
LIN {X 0,Y 436.009,Z 942.11,A -85,B 0,C 180,E1 10451.685,E2 10451.685} C_VEL
LIN {X 0,Y 441.236,Z 919.625,A -85,B 0,C 180,E1 10451.218,E2 10451.218} C_VEL
LIN {X 0,Y 446.359,Z 890.373,A -85,B 0,C 180,E1 10450.74,E2 10450.74} C_VEL
LIN {X 0,Y 452.159,Z 838.553,A -85,B 0,C 180,E1 10450.005,E2 10450.005} C_VEL
LIN {X 0,Y 454.022,Z 820.94,A -85,B 0,C 180,E1 10449.76,E2 10449.76} C_VEL
LIN {X 0,Y 454.661,Z 813.413,A -85,B 0,C 180,E1 10449.534,E2 10449.534} C_VEL
LIN {X 0,Y 455.788,Z 793.909,A -85,B 0,C 180,E1 10448.48,E2 10448.48} C_VEL
LIN {X 0,Y 456.382,Z 787.436,A -85,B 0,C 180,E1 10448.297,E2 10448.297} C_VEL
LIN {X 0,Y 465.49,Z 704.125,A -85,B 0,C 180,E1 10447.157,E2 10447.157} C_VEL
LIN {X 0,Y 464.124,Z 700.987,A -85,B 0,C 180,E1 10445.068,E2 10445.068} C_VEL
LIN {X 0,Y 462.964,Z 696.946,A -85,B 0,C 180,E1 10440.619,E2 10440.619} C_VEL
LIN {X 0,Y 462.974,Z 697.16,A -85,B 0,C 180,E1 10439.381,E2 10439.381} C_VEL
LIN {X 0,Y 464.503,Z 701.859,A -85,B 0,C 180,E1 10434.689,E2 10434.689} C_VEL
LIN {X 0,Y 465.558,Z 704.535,A -85,B 0,C 180,E1 10433.141,E2 10433.141} C_VEL
LIN {X 0,Y 445.12,Z 891.218,A -85,B 0,C 180,E1 10430.569,E2 10430.569} C_VEL
LIN {X 0,Y 441.032,Z 916.843,A -85,B 0,C 180,E1 10430.176,E2 10430.176} C_VEL
LIN {X 0,Y 434.683,Z 944.953,A -85,B 0,C 180,E1 10429.687,E2 10429.687} C_VEL
LIN {X 0,Y 428.543,Z 966.759,A -85,B 0,C 180,E1 10429.215,E2 10429.215} C_VEL
LIN {X 0,Y 421.7,Z 987.497,A -85,B 0,C 180,E1 10428.665,E2 10428.665} C_VEL
LIN {X 0,Y 413.6,Z 1008.86,A -85,B 0,C 180,E1 10427.977,E2 10427.977} C_VEL
LIN {X 0,Y 402.37,Z 1034.641,A -85,B 0,C 180,E1 10426.951,E2 10426.951} C_VEL
LIN {X 0,Y 391.156,Z 1056.932,A -85,B 0,C 180,E1 10425.853,E2 10425.853} C_VEL
LIN {X 0,Y 380.881,Z 1075.436,A -85,B 0,C 180,E1 10424.758,E2 10424.758} C_VEL
LIN {X 0,Y 369.922,Z 1093.462,A -85,B 0,C 180,E1 10423.512,E2 10423.512} C_VEL
LIN {X 0,Y 356.903,Z 1113.15,A -85,B 0,C 180,E1 10421.882,E2 10421.882} C_VEL
LIN {X 0,Y 340.798,Z 1135.203,A -85,B 0,C 180,E1 10419.633,E2 10419.633} C_VEL
LIN {X 0,Y 327.387,Z 1152.071,A -85,B 0,C 180,E1 10417.513,E2 10417.513} C_VEL
LIN {X 0,Y 314.835,Z 1166.885,A -85,B 0,C 180,E1 10415.286,E2 10415.286} C_VEL
LIN {X 0,Y 301.718,Z 1181.505,A -85,B 0,C 180,E1 10412.654,E2 10412.654} C_VEL
LIN {X 0,Y 285.3,Z 1198.796,A -85,B 0,C 180,E1 10408.788,E2 10408.788} C_VEL
LIN {X 0,Y 271.792,Z 1212.234,A -85,B 0,C 180,E1 10404.977,E2 10404.977} C_VEL
LIN {X 0,Y 260.541,Z 1223.154,A -85,B 0,C 180,E1 10401.187,E2 10401.187} C_VEL
LIN {X 0,Y 249.751,Z 1233.529,A -85,B 0,C 180,E1 10396.785,E2 10396.785} C_VEL
LIN {X 0,Y 238.387,Z 1244.615,A -85,B 0,C 180,E1 10390.88,E2 10390.88} C_VEL
LIN {X 0,Y 229.69,Z 1253.347,A -85,B 0,C 180,E1 10384.781,E2 10384.781} C_VEL
LIN {X 0,Y 224.128,Z 1259.479,A -85,B 0,C 180,E1 10379.401,E2 10379.401} C_VEL
LIN {X 0,Y 220.148,Z 1264.508,A -85,B 0,C 180,E1 10373.854,E2 10373.854} C_VEL
LIN {X 0,Y 217.639,Z 1268.461,A -85,B 0,C 180,E1 10368.216,E2 10368.216} C_VEL
LIN {X 0,Y 216.378,Z 1271.356,A -85,B 0,C 180,E1 10362.556,E2 10362.556} C_VEL
LIN {X 0,Y 216.03,Z 1273.203,A -85,B 0,C 180,E1 10356.924,E2 10356.924} C_VEL
LIN {X 0,Y 216.023,Z 1273.948,A -85,B 0,C 180,E1 10351.869,E2 10351.869} C_VEL
LIN {X 0,Y 216.018,Z 1273.875,A -85,B 0,C 180,E1 10347.359,E2 10347.359} C_VEL
LIN {X 0,Y 216.034,Z 1273.129,A -85,B 0,C 180,E1 10342.834,E2 10342.834} C_VEL
LIN {X 0,Y 216.375,Z 1271.352,A -85,B 0,C 180,E1 10337.469,E2 10337.469} C_VEL
LIN {X 0,Y 217.631,Z 1268.455,A -85,B 0,C 180,E1 10331.809,E2 10331.809} C_VEL
LIN {X 0,Y 220.132,Z 1264.501,A -85,B 0,C 180,E1 10326.17,E2 10326.17} C_VEL
LIN {X 0,Y 224.105,Z 1259.47,A -85,B 0,C 180,E1 10320.623,E2 10320.623} C_VEL
LIN {X 0,Y 229.962,Z 1253.019,A -85,B 0,C 180,E1 10314.991,E2 10314.991} C_VEL
LIN {X 0,Y 239.543,Z 1243.414,A -85,B 0,C 180,E1 10308.436,E2 10308.436} C_VEL
LIN {X 0,Y 250.18,Z 1233.036,A -85,B 0,C 180,E1 10303.016,E2 10303.016} C_VEL
LIN {X 0,Y 260.483,Z 1223.129,A -85,B 0,C 180,E1 10298.83,E2 10298.83} C_VEL
LIN {X 0,Y 271.99,Z 1211.949,A -85,B 0,C 180,E1 10294.957,E2 10294.957} C_VEL
LIN {X 0,Y 286.771,Z 1197.242,A -85,B 0,C 180,E1 10290.834,E2 10290.834} C_VEL
LIN {X 0,Y 302.349,Z 1180.658,A -85,B 0,C 180,E1 10287.202,E2 10287.202} C_VEL
LIN {X 0,Y 314.754,Z 1166.81,A -85,B 0,C 180,E1 10284.722,E2 10284.722} C_VEL
LIN {X 0,Y 327.303,Z 1151.986,A -85,B 0,C 180,E1 10282.493,E2 10282.493} C_VEL
LIN {X 0,Y 340.711,Z 1135.104,A -85,B 0,C 180,E1 10280.372,E2 10280.372} C_VEL
LIN {X 0,Y 356.785,Z 1113.059,A -85,B 0,C 180,E1 10278.124,E2 10278.124} C_VEL
LIN {X 0,Y 369.214,Z 1094.284,A -85,B 0,C 180,E1 10276.563,E2 10276.563} C_VEL
LIN {X 0,Y 380.355,Z 1076,A -85,B 0,C 180,E1 10275.29,E2 10275.29} C_VEL
LIN {X 0,Y 390.788,Z 1057.243,A -85,B 0,C 180,E1 10274.174,E2 10274.174} C_VEL
LIN {X 0,Y 402.274,Z 1034.426,A -85,B 0,C 180,E1 10273.048,E2 10273.048} C_VEL
LIN {X 0,Y 413.504,Z 1008.579,A -85,B 0,C 180,E1 10272.021,E2 10272.021} C_VEL
LIN {X 0,Y 421.559,Z 987.294,A -85,B 0,C 180,E1 10271.336,E2 10271.336} C_VEL
LIN {X 0,Y 428.447,Z 966.371,A -85,B 0,C 180,E1 10270.782,E2 10270.782} C_VEL
LIN {X 0,Y 434.751,Z 943.869,A -85,B 0,C 180,E1 10270.298,E2 10270.298} C_VEL
LIN {X 0,Y 441.346,Z 913.759,A -85,B 0,C 180,E1 10269.781,E2 10269.781} C_VEL
LIN {X 0,Y 445.01,Z 890.317,A -85,B 0,C 180,E1 10269.423,E2 10269.423} C_VEL
LIN {X 0,Y 465.35,Z 704.208,A -85,B 0,C 180,E1 10266.856,E2 10266.856} C_VEL
LIN {X 0,Y 463.908,Z 700.915,A -85,B 0,C 180,E1 10264.698,E2 10264.698} C_VEL
LIN {X 0,Y 462.724,Z 697.179,A -85,B 0,C 180,E1 10260.867,E2 10260.867} C_VEL
LIN {X 0,Y 462.721,Z 697.043,A -85,B 0,C 180,E1 10258.762,E2 10258.762} C_VEL
LIN {X 0,Y 464.273,Z 701.707,A -85,B 0,C 180,E1 10254.175,E2 10254.175} C_VEL
LIN {X 0,Y 465.252,Z 704.147,A -85,B 0,C 180,E1 10252.742,E2 10252.742} C_VEL
LIN {X 0,Y 445.263,Z 886.335,A -85,B 0,C 180,E1 10250.239,E2 10250.239} C_VEL
LIN {X 0,Y 441.19,Z 911.783,A -85,B 0,C 180,E1 10249.851,E2 10249.851} C_VEL
LIN {X 0,Y 434.954,Z 939.621,A -85,B 0,C 180,E1 10249.315,E2 10249.315} C_VEL
LIN {X 0,Y 428.828,Z 961.553,A -85,B 0,C 180,E1 10248.781,E2 10248.781} C_VEL
LIN {X 0,Y 421.868,Z 982.718,A -85,B 0,C 180,E1 10248.155,E2 10248.155} C_VEL
LIN {X 0,Y 413.404,Z 1005.002,A -85,B 0,C 180,E1 10247.36,E2 10247.36} C_VEL
LIN {X 0,Y 401.934,Z 1030.875,A -85,B 0,C 180,E1 10246.234,E2 10246.234} C_VEL
LIN {X 0,Y 391.927,Z 1050.688,A -85,B 0,C 180,E1 10245.18,E2 10245.18} C_VEL
LIN {X 0,Y 381.523,Z 1069.29,A -85,B 0,C 180,E1 10244.027,E2 10244.027} C_VEL
LIN {X 0,Y 370.2,Z 1087.766,A -85,B 0,C 180,E1 10242.67,E2 10242.67} C_VEL
LIN {X 0,Y 356.049,Z 1108.865,A -85,B 0,C 180,E1 10240.818,E2 10240.818} C_VEL
LIN {X 0,Y 341.253,Z 1128.564,A -85,B 0,C 180,E1 10238.681,E2 10238.681} C_VEL
LIN {X 0,Y 328.781,Z 1143.974,A -85,B 0,C 180,E1 10236.672,E2 10236.672} C_VEL
LIN {X 0,Y 316.721,Z 1157.929,A -85,B 0,C 180,E1 10234.516,E2 10234.516} C_VEL
LIN {X 0,Y 303.715,Z 1172.112,A -85,B 0,C 180,E1 10231.897,E2 10231.897} C_VEL
LIN {X 0,Y 288.068,Z 1188.212,A -85,B 0,C 180,E1 10228.232,E2 10228.232} C_VEL
LIN {X 0,Y 274.216,Z 1201.522,A -85,B 0,C 180,E1 10224.382,E2 10224.382} C_VEL
LIN {X 0,Y 262.698,Z 1212.227,A -85,B 0,C 180,E1 10220.574,E2 10220.574} C_VEL
LIN {X 0,Y 252.052,Z 1221.914,A -85,B 0,C 180,E1 10216.349,E2 10216.349} C_VEL
LIN {X 0,Y 240.716,Z 1232.281,A -85,B 0,C 180,E1 10210.687,E2 10210.687} C_VEL
LIN {X 0,Y 231.356,Z 1240.835,A -85,B 0,C 180,E1 10204.467,E2 10204.467} C_VEL
LIN {X 0,Y 225.501,Z 1246.598,A -85,B 0,C 180,E1 10199.13,E2 10199.13} C_VEL
LIN {X 0,Y 221.063,Z 1251.409,A -85,B 0,C 180,E1 10193.441,E2 10193.441} C_VEL
LIN {X 0,Y 218.275,Z 1254.984,A -85,B 0,C 180,E1 10187.86,E2 10187.86} C_VEL
LIN {X 0,Y 216.714,Z 1257.669,A -85,B 0,C 180,E1 10181.97,E2 10181.97} C_VEL
LIN {X 0,Y 216.129,Z 1259.365,A -85,B 0,C 180,E1 10175.829,E2 10175.829} C_VEL
LIN {X 0,Y 216.011,Z 1259.903,A -85,B 0,C 180,E1 10170.253,E2 10170.253} C_VEL
LIN {X 0,Y 216.105,Z 1259.506,A -85,B 0,C 180,E1 10164.679,E2 10164.679} C_VEL
LIN {X 0,Y 216.651,Z 1257.82,A -85,B 0,C 180,E1 10158.272,E2 10158.272} C_VEL
LIN {X 0,Y 218.157,Z 1255.196,A -85,B 0,C 180,E1 10152.381,E2 10152.381} C_VEL
LIN {X 0,Y 221.034,Z 1251.483,A -85,B 0,C 180,E1 10146.53,E2 10146.53} C_VEL
LIN {X 0,Y 225.495,Z 1246.648,A -85,B 0,C 180,E1 10140.795,E2 10140.795} C_VEL
LIN {X 0,Y 231.613,Z 1240.65,A -85,B 0,C 180,E1 10135.249,E2 10135.249} C_VEL
LIN {X 0,Y 241.101,Z 1231.988,A -85,B 0,C 180,E1 10129.007,E2 10129.007} C_VEL
LIN {X 0,Y 252.239,Z 1221.821,A -85,B 0,C 180,E1 10123.485,E2 10123.485} C_VEL
LIN {X 0,Y 262.615,Z 1212.392,A -85,B 0,C 180,E1 10119.372,E2 10119.372} C_VEL
LIN {X 0,Y 274.13,Z 1201.704,A -85,B 0,C 180,E1 10115.56,E2 10115.56} C_VEL
LIN {X 0,Y 288.646,Z 1187.788,A -85,B 0,C 180,E1 10111.539,E2 10111.539} C_VEL
LIN {X 0,Y 303.637,Z 1172.355,A -85,B 0,C 180,E1 10108.038,E2 10108.038} C_VEL
LIN {X 0,Y 316.646,Z 1158.191,A -85,B 0,C 180,E1 10105.417,E2 10105.417} C_VEL
LIN {X 0,Y 329.479,Z 1143.341,A -85,B 0,C 180,E1 10103.13,E2 10103.13} C_VEL
LIN {X 0,Y 342.777,Z 1126.864,A -85,B 0,C 180,E1 10101.009,E2 10101.009} C_VEL
LIN {X 0,Y 358.947,Z 1104.885,A -85,B 0,C 180,E1 10098.705,E2 10098.705} C_VEL
LIN {X 0,Y 370.989,Z 1086.836,A -85,B 0,C 180,E1 10097.154,E2 10097.154} C_VEL
LIN {X 0,Y 381.989,Z 1068.845,A -85,B 0,C 180,E1 10095.84,E2 10095.84} C_VEL
LIN {X 0,Y 392.753,Z 1049.538,A -85,B 0,C 180,E1 10094.652,E2 10094.652} C_VEL
LIN {X 0,Y 404.46,Z 1026.111,A -85,B 0,C 180,E1 10093.438,E2 10093.438} C_VEL
LIN {X 0,Y 414.707,Z 1002.238,A -85,B 0,C 180,E1 10092.436,E2 10092.436} C_VEL
LIN {X 0,Y 422.318,Z 982.055,A -85,B 0,C 180,E1 10091.727,E2 10091.727} C_VEL
LIN {X 0,Y 429.035,Z 961.598,A -85,B 0,C 180,E1 10091.124,E2 10091.124} C_VEL
LIN {X 0,Y 435.223,Z 939.439,A -85,B 0,C 180,E1 10090.584,E2 10090.584} C_VEL
LIN {X 0,Y 441.514,Z 911.199,A -85,B 0,C 180,E1 10090.043,E2 10090.043} C_VEL
LIN {X 0,Y 445.498,Z 886.278,A -85,B 0,C 180,E1 10089.665,E2 10089.665} C_VEL
LIN {X 0,Y 456.382,Z 787.436,A -85,B 0,C 180,E1 10088.297,E2 10088.297} C_VEL
LIN {X 0,Y 457.062,Z 779.912,A -85,B 0,C 180,E1 10088.071,E2 10088.071} C_VEL
LIN {X 0,Y 458.401,Z 760.412,A -85,B 0,C 180,E1 10087.026,E2 10087.026} C_VEL
LIN {X 0,Y 459.032,Z 753.938,A -85,B 0,C 180,E1 10086.847,E2 10086.847} C_VEL
LIN {X 0,Y 463.829,Z 710.789,A -85,B 0,C 180,E1 10086.25,E2 10086.25} C_VEL
LIN {X 0,Y 463.007,Z 708.771,A -85,B 0,C 180,E1 10084.831,E2 10084.831} C_VEL
LIN {X 0,Y 461.983,Z 704.89,A -85,B 0,C 180,E1 10080.496,E2 10080.496} C_VEL
LIN {X 0,Y 461.989,Z 705.182,A -85,B 0,C 180,E1 10079.38,E2 10079.38} C_VEL
LIN {X 0,Y 463.407,Z 709.66,A -85,B 0,C 180,E1 10074.863,E2 10074.863} C_VEL
LIN {X 0,Y 463.888,Z 711.234,A -85,B 0,C 180,E1 10074.035,E2 10074.035} C_VEL
LIN {X 0,Y 443.865,Z 891.023,A -85,B 0,C 180,E1 10071.593,E2 10071.593} C_VEL
LIN {X 0,Y 439.673,Z 916.92,A -85,B 0,C 180,E1 10071.205,E2 10071.205} C_VEL
LIN {X 0,Y 433.254,Z 944.917,A -85,B 0,C 180,E1 10070.731,E2 10070.731} C_VEL
LIN {X 0,Y 427.106,Z 966.503,A -85,B 0,C 180,E1 10070.28,E2 10070.28} C_VEL
LIN {X 0,Y 420.184,Z 987.238,A -85,B 0,C 180,E1 10069.748,E2 10069.748} C_VEL
LIN {X 0,Y 412.074,Z 1008.374,A -85,B 0,C 180,E1 10069.09,E2 10069.09} C_VEL
LIN {X 0,Y 400.607,Z 1034.379,A -85,B 0,C 180,E1 10068.088,E2 10068.088} C_VEL
LIN {X 0,Y 389.402,Z 1056.359,A -85,B 0,C 180,E1 10067.039,E2 10067.039} C_VEL
LIN {X 0,Y 378.593,Z 1075.522,A -85,B 0,C 180,E1 10065.938,E2 10065.938} C_VEL
LIN {X 0,Y 367.038,Z 1094.172,A -85,B 0,C 180,E1 10064.674,E2 10064.674} C_VEL
LIN {X 0,Y 352.543,Z 1115.608,A -85,B 0,C 180,E1 10062.917,E2 10062.917} C_VEL
LIN {X 0,Y 336.761,Z 1136.471,A -85,B 0,C 180,E1 10060.781,E2 10060.781} C_VEL
LIN {X 0,Y 323.886,Z 1152.269,A -85,B 0,C 180,E1 10058.814,E2 10058.814} C_VEL
LIN {X 0,Y 311.419,Z 1166.612,A -85,B 0,C 180,E1 10056.689,E2 10056.689} C_VEL
LIN {X 0,Y 297.943,Z 1181.231,A -85,B 0,C 180,E1 10054.093,E2 10054.093} C_VEL
LIN {X 0,Y 281.023,Z 1198.521,A -85,B 0,C 180,E1 10050.259,E2 10050.259} C_VEL
LIN {X 0,Y 267.304,Z 1211.706,A -85,B 0,C 180,E1 10046.542,E2 10046.542} C_VEL
LIN {X 0,Y 255.332,Z 1222.879,A -85,B 0,C 180,E1 10042.663,E2 10042.663} C_VEL
LIN {X 0,Y 244.038,Z 1233.253,A -85,B 0,C 180,E1 10038.232,E2 10038.232} C_VEL
LIN {X 0,Y 231.868,Z 1244.522,A -85,B 0,C 180,E1 10032.122,E2 10032.122} C_VEL
LIN {X 0,Y 222.837,Z 1253.072,A -85,B 0,C 180,E1 10026.014,E2 10026.014} C_VEL
LIN {X 0,Y 216.817,Z 1259.275,A -85,B 0,C 180,E1 10020.414,E2 10020.414} C_VEL
LIN {X 0,Y 212.607,Z 1264.195,A -85,B 0,C 180,E1 10014.813,E2 10014.813} C_VEL
LIN {X 0,Y 209.849,Z 1268.191,A -85,B 0,C 180,E1 10008.917,E2 10008.917} C_VEL
LIN {X 0,Y 208.401,Z 1271.209,A -85,B 0,C 180,E1 10002.763,E2 10002.763} C_VEL
LIN {X 0,Y 208.023,Z 1273.154,A -85,B 0,C 180,E1 9996.359,E2 9996.359} C_VEL
LIN {X 0,Y 208.007,Z 1273.756,A -85,B 0,C 180,E1 9991.114,E2 9991.114} C_VEL
LIN {X 0,Y 208.013,Z 1273.489,A -85,B 0,C 180,E1 9985.878,E2 9985.878} C_VEL
LIN {X 0,Y 208.083,Z 1272.355,A -85,B 0,C 180,E1 9980.61,E2 9980.61} C_VEL
LIN {X 0,Y 208.887,Z 1270.002,A -85,B 0,C 180,E1 9974.465,E2 9974.465} C_VEL
LIN {X 0,Y 211.632,Z 1265.521,A -85,B 0,C 180,E1 9966.927,E2 9966.927} C_VEL
LIN {X 0,Y 216.152,Z 1259.988,A -85,B 0,C 180,E1 9960.348,E2 9960.348} C_VEL
LIN {X 0,Y 221.859,Z 1253.997,A -85,B 0,C 180,E1 9954.786,E2 9954.786} C_VEL
LIN {X 0,Y 229.498,Z 1246.6,A -85,B 0,C 180,E1 9949.297,E2 9949.297} C_VEL
LIN {X 0,Y 240.756,Z 1236.299,A -85,B 0,C 180,E1 9943.257,E2 9943.257} C_VEL
LIN {X 0,Y 253.569,Z 1224.431,A -85,B 0,C 180,E1 9937.961,E2 9937.961} C_VEL
LIN {X 0,Y 265.368,Z 1213.427,A -85,B 0,C 180,E1 9934.032,E2 9934.032} C_VEL
LIN {X 0,Y 277.574,Z 1201.71,A -85,B 0,C 180,E1 9930.602,E2 9930.602} C_VEL
LIN {X 0,Y 291.37,Z 1187.936,A -85,B 0,C 180,E1 9927.303,E2 9927.303} C_VEL
LIN {X 0,Y 309.053,Z 1169.106,A -85,B 0,C 180,E1 9923.738,E2 9923.738} C_VEL
LIN {X 0,Y 322.612,Z 1153.585,A -85,B 0,C 180,E1 9921.384,E2 9921.384} C_VEL
LIN {X 0,Y 335.303,Z 1138.086,A -85,B 0,C 180,E1 9919.421,E2 9919.421} C_VEL
LIN {X 0,Y 348.246,Z 1121.136,A -85,B 0,C 180,E1 9917.626,E2 9917.626} C_VEL
LIN {X 0,Y 363.511,Z 1099.402,A -85,B 0,C 180,E1 9915.731,E2 9915.731} C_VEL
LIN {X 0,Y 377.059,Z 1077.773,A -85,B 0,C 180,E1 9914.217,E2 9914.217} C_VEL
LIN {X 0,Y 387.698,Z 1059.108,A -85,B 0,C 180,E1 9913.118,E2 9913.118} C_VEL
LIN {X 0,Y 397.805,Z 1039.589,A -85,B 0,C 180,E1 9912.154,E2 9912.154} C_VEL
LIN {X 0,Y 408.204,Z 1017.163,A -85,B 0,C 180,E1 9911.231,E2 9911.231} C_VEL
LIN {X 0,Y 418.709,Z 990.763,A -85,B 0,C 180,E1 9910.359,E2 9910.359} C_VEL
LIN {X 0,Y 426.083,Z 969.067,A -85,B 0,C 180,E1 9909.786,E2 9909.786} C_VEL
LIN {X 0,Y 432.207,Z 947.992,A -85,B 0,C 180,E1 9909.333,E2 9909.333} C_VEL
LIN {X 0,Y 437.561,Z 925.818,A -85,B 0,C 180,E1 9908.944,E2 9908.944} C_VEL
LIN {X 0,Y 442.738,Z 897.875,A -85,B 0,C 180,E1 9908.509,E2 9908.509} C_VEL
LIN {X 0,Y 448.121,Z 852.047,A -85,B 0,C 180,E1 9907.874,E2 9907.874} C_VEL
LIN {X 0,Y 463.664,Z 710.858,A -85,B 0,C 180,E1 9905.941,E2 9905.941} C_VEL
LIN {X 0,Y 462.788,Z 708.691,A -85,B 0,C 180,E1 9904.461,E2 9904.461} C_VEL
LIN {X 0,Y 461.719,Z 704.87,A -85,B 0,C 180,E1 9900.372,E2 9900.372} C_VEL
LIN {X 0,Y 461.735,Z 705.072,A -85,B 0,C 180,E1 9898.759,E2 9898.759} C_VEL
LIN {X 0,Y 463.202,Z 709.591,A -85,B 0,C 180,E1 9894.301,E2 9894.301} C_VEL
LIN {X 0,Y 463.58,Z 710.941,A -85,B 0,C 180,E1 9893.635,E2 9893.635} C_VEL
LIN {X 0,Y 443.962,Z 886.727,A -85,B 0,C 180,E1 9891.256,E2 9891.256} C_VEL
LIN {X 0,Y 439.735,Z 912.71,A -85,B 0,C 180,E1 9890.868,E2 9890.868} C_VEL
LIN {X 0,Y 433.482,Z 940.112,A -85,B 0,C 180,E1 9890.352,E2 9890.352} C_VEL
LIN {X 0,Y 427.338,Z 961.826,A -85,B 0,C 180,E1 9889.837,E2 9889.837} C_VEL
LIN {X 0,Y 420.742,Z 981.713,A -85,B 0,C 180,E1 9889.269,E2 9889.269} C_VEL
LIN {X 0,Y 413.061,Z 1001.904,A -85,B 0,C 180,E1 9888.582,E2 9888.582} C_VEL
LIN {X 0,Y 402.76,Z 1025.655,A -85,B 0,C 180,E1 9887.616,E2 9887.616} C_VEL
LIN {X 0,Y 390.806,Z 1049.352,A -85,B 0,C 180,E1 9886.426,E2 9886.426} C_VEL
LIN {X 0,Y 379.703,Z 1068.991,A -85,B 0,C 180,E1 9885.247,E2 9885.247} C_VEL
LIN {X 0,Y 368.822,Z 1086.535,A -85,B 0,C 180,E1 9883.998,E2 9883.998} C_VEL
LIN {X 0,Y 356.907,Z 1104.137,A -85,B 0,C 180,E1 9882.531,E2 9882.531} C_VEL
LIN {X 0,Y 341.186,Z 1125.335,A -85,B 0,C 180,E1 9880.391,E2 9880.391} C_VEL
LIN {X 0,Y 327.167,Z 1142.422,A -85,B 0,C 180,E1 9878.263,E2 9878.263} C_VEL
LIN {X 0,Y 314.006,Z 1157.371,A -85,B 0,C 180,E1 9876.021,E2 9876.021} C_VEL
LIN {X 0,Y 301.349,Z 1170.871,A -85,B 0,C 180,E1 9873.594,E2 9873.594} C_VEL
LIN {X 0,Y 287.868,Z 1184.447,A -85,B 0,C 180,E1 9870.648,E2 9870.648} C_VEL
LIN {X 0,Y 271.325,Z 1200.114,A -85,B 0,C 180,E1 9866.371,E2 9866.371} C_VEL
LIN {X 0,Y 258.264,Z 1211.805,A -85,B 0,C 180,E1 9862.287,E2 9862.287} C_VEL
LIN {X 0,Y 247.378,Z 1221.316,A -85,B 0,C 180,E1 9858.17,E2 9858.17} C_VEL
LIN {X 0,Y 237.062,Z 1230.205,A -85,B 0,C 180,E1 9853.415,E2 9853.415} C_VEL
LIN {X 0,Y 226.19,Z 1239.719,A -85,B 0,C 180,E1 9846.857,E2 9846.857} C_VEL
LIN {X 0,Y 218.61,Z 1246.585,A -85,B 0,C 180,E1 9840.495,E2 9840.495} C_VEL
LIN {X 0,Y 213.726,Z 1251.482,A -85,B 0,C 180,E1 9834.591,E2 9834.591} C_VEL
LIN {X 0,Y 210.629,Z 1255.1,A -85,B 0,C 180,E1 9828.818,E2 9828.818} C_VEL
LIN {X 0,Y 208.912,Z 1257.719,A -85,B 0,C 180,E1 9822.986,E2 9822.986} C_VEL
LIN {X 0,Y 208.189,Z 1259.434,A -85,B 0,C 180,E1 9816.883,E2 9816.883} C_VEL
LIN {X 0,Y 208.024,Z 1260.076,A -85,B 0,C 180,E1 9811.364,E2 9811.364} C_VEL
LIN {X 0,Y 208.076,Z 1259.872,A -85,B 0,C 180,E1 9805.854,E2 9805.854} C_VEL
LIN {X 0,Y 208.423,Z 1258.756,A -85,B 0,C 180,E1 9800.043,E2 9800.043} C_VEL
LIN {X 0,Y 209.911,Z 1256.226,A -85,B 0,C 180,E1 9793.096,E2 9793.096} C_VEL
LIN {X 0,Y 213.194,Z 1252.111,A -85,B 0,C 180,E1 9786.144,E2 9786.144} C_VEL
LIN {X 0,Y 217.924,Z 1247.287,A -85,B 0,C 180,E1 9780.133,E2 9780.133} C_VEL
LIN {X 0,Y 224.164,Z 1241.507,A -85,B 0,C 180,E1 9774.547,E2 9774.547} C_VEL
LIN {X 0,Y 232.289,Z 1234.395,A -85,B 0,C 180,E1 9769.123,E2 9769.123} C_VEL
LIN {X 0,Y 245.049,Z 1223.436,A -85,B 0,C 180,E1 9762.726,E2 9762.726} C_VEL
LIN {X 0,Y 256.827,Z 1213.167,A -85,B 0,C 180,E1 9758.134,E2 9758.134} C_VEL
LIN {X 0,Y 268.12,Z 1203.099,A -85,B 0,C 180,E1 9754.483,E2 9754.483} C_VEL
LIN {X 0,Y 280.334,Z 1191.799,A -85,B 0,C 180,E1 9751.114,E2 9751.114} C_VEL
LIN {X 0,Y 295.523,Z 1177.093,A -85,B 0,C 180,E1 9747.555,E2 9747.555} C_VEL
LIN {X 0,Y 311.669,Z 1160.125,A -85,B 0,C 180,E1 9744.326,E2 9744.326} C_VEL
LIN {X 0,Y 324.754,Z 1145.436,A -85,B 0,C 180,E1 9742.053,E2 9742.053} C_VEL
LIN {X 0,Y 337.095,Z 1130.614,A -85,B 0,C 180,E1 9740.126,E2 9740.126} C_VEL
LIN {X 0,Y 349.746,Z 1114.266,A -85,B 0,C 180,E1 9738.33,E2 9738.33} C_VEL
LIN {X 0,Y 364.889,Z 1092.962,A -85,B 0,C 180,E1 9736.394,E2 9736.394} C_VEL
LIN {X 0,Y 377.939,Z 1072.314,A -85,B 0,C 180,E1 9734.87,E2 9734.87} C_VEL
LIN {X 0,Y 388.582,Z 1053.824,A -85,B 0,C 180,E1 9733.728,E2 9733.728} C_VEL
LIN {X 0,Y 398.237,Z 1035.293,A -85,B 0,C 180,E1 9732.742,E2 9732.742} C_VEL
LIN {X 0,Y 407.156,Z 1016.304,A -85,B 0,C 180,E1 9731.885,E2 9731.885} C_VEL
LIN {X 0,Y 416.658,Z 993.506,A -85,B 0,C 180,E1 9731.019,E2 9731.019} C_VEL
LIN {X 0,Y 425.963,Z 967.008,A -85,B 0,C 180,E1 9730.205,E2 9730.205} C_VEL
LIN {X 0,Y 432.557,Z 944.451,A -85,B 0,C 180,E1 9729.645,E2 9729.645} C_VEL
LIN {X 0,Y 437.762,Z 923.003,A -85,B 0,C 180,E1 9729.214,E2 9729.214} C_VEL
LIN {X 0,Y 442.282,Z 899.609,A -85,B 0,C 180,E1 9728.836,E2 9728.836} C_VEL
LIN {X 0,Y 446.952,Z 863.772,A -85,B 0,C 180,E1 9728.33,E2 9728.33} C_VEL
LIN {X 0,Y 459.032,Z 753.938,A -85,B 0,C 180,E1 9726.847,E2 9726.847} C_VEL
LIN {X 0,Y 459.757,Z 746.417,A -85,B 0,C 180,E1 9726.624,E2 9726.624} C_VEL
LIN {X 0,Y 461.3,Z 726.932,A -85,B 0,C 180,E1 9725.585,E2 9725.585} C_VEL
LIN {X 0,Y 461.965,Z 720.462,A -85,B 0,C 180,E1 9725.408,E2 9725.408} C_VEL
LIN {X 0,Y 462.295,Z 717.367,A -85,B 0,C 180,E1 9725.336,E2 9725.336} C_VEL
LIN {X 0,Y 461.008,Z 712.831,A -85,B 0,C 180,E1 9720.497,E2 9720.497} C_VEL
LIN {X 0,Y 461.004,Z 713.203,A -85,B 0,C 180,E1 9719.379,E2 9719.379} C_VEL
LIN {X 0,Y 462.348,Z 717.568,A -85,B 0,C 180,E1 9714.975,E2 9714.975} C_VEL
LIN {X 0,Y 462.242,Z 718.725,A -85,B 0,C 180,E1 9714.925,E2 9714.925} C_VEL
LIN {X 0,Y 442.759,Z 890.78,A -85,B 0,C 180,E1 9712.624,E2 9712.624} C_VEL
LIN {X 0,Y 438.485,Z 916.834,A -85,B 0,C 180,E1 9712.242,E2 9712.242} C_VEL
LIN {X 0,Y 432.013,Z 944.724,A -85,B 0,C 180,E1 9711.785,E2 9711.785} C_VEL
LIN {X 0,Y 425.816,Z 966.247,A -85,B 0,C 180,E1 9711.351,E2 9711.351} C_VEL
LIN {X 0,Y 418.95,Z 986.616,A -85,B 0,C 180,E1 9710.848,E2 9710.848} C_VEL
LIN {X 0,Y 410.938,Z 1007.318,A -85,B 0,C 180,E1 9710.229,E2 9710.229} C_VEL
LIN {X 0,Y 399.918,Z 1032.297,A -85,B 0,C 180,E1 9709.311,E2 9709.311} C_VEL
LIN {X 0,Y 387.692,Z 1056.013,A -85,B 0,C 180,E1 9708.223,E2 9708.223} C_VEL
LIN {X 0,Y 377.07,Z 1074.603,A -85,B 0,C 180,E1 9707.192,E2 9707.192} C_VEL
LIN {X 0,Y 365.414,Z 1093.185,A -85,B 0,C 180,E1 9705.975,E2 9705.975} C_VEL
LIN {X 0,Y 352.348,Z 1112.269,A -85,B 0,C 180,E1 9704.473,E2 9704.473} C_VEL
LIN {X 0,Y 335.337,Z 1134.704,A -85,B 0,C 180,E1 9702.294,E2 9702.294} C_VEL
LIN {X 0,Y 321.772,Z 1151.059,A -85,B 0,C 180,E1 9700.329,E2 9700.329} C_VEL
LIN {X 0,Y 308.977,Z 1165.481,A -85,B 0,C 180,E1 9698.258,E2 9698.258} C_VEL
LIN {X 0,Y 295.842,Z 1179.413,A -85,B 0,C 180,E1 9695.861,E2 9695.861} C_VEL
LIN {X 0,Y 281.875,Z 1193.423,A -85,B 0,C 180,E1 9692.933,E2 9692.933} C_VEL
LIN {X 0,Y 264.043,Z 1210.26,A -85,B 0,C 180,E1 9688.447,E2 9688.447} C_VEL
LIN {X 0,Y 250.996,Z 1221.99,A -85,B 0,C 180,E1 9684.435,E2 9684.435} C_VEL
LIN {X 0,Y 239.558,Z 1232.036,A -85,B 0,C 180,E1 9680.187,E2 9680.187} C_VEL
LIN {X 0,Y 228.578,Z 1241.634,A -85,B 0,C 180,E1 9675.138,E2 9675.138} C_VEL
LIN {X 0,Y 216.978,Z 1251.993,A -85,B 0,C 180,E1 9668,E2 9668} C_VEL
LIN {X 0,Y 209.978,Z 1258.667,A -85,B 0,C 180,E1 9661.921,E2 9661.921} C_VEL
LIN {X 0,Y 205.428,Z 1263.532,A -85,B 0,C 180,E1 9656.303,E2 9656.303} C_VEL
LIN {X 0,Y 202.408,Z 1267.418,A -85,B 0,C 180,E1 9650.545,E2 9650.545} C_VEL
LIN {X 0,Y 200.712,Z 1270.341,A -85,B 0,C 180,E1 9644.731,E2 9644.731} C_VEL
LIN {X 0,Y 200.08,Z 1272.238,A -85,B 0,C 180,E1 9639.215,E2 9639.215} C_VEL
LIN {X 0,Y 200.02,Z 1273.252,A -85,B 0,C 180,E1 9634.026,E2 9634.026} C_VEL
LIN {X 0,Y 200.011,Z 1273.492,A -85,B 0,C 180,E1 9628.867,E2 9628.867} C_VEL
LIN {X 0,Y 200.029,Z 1272.887,A -85,B 0,C 180,E1 9623.412,E2 9623.412} C_VEL
LIN {X 0,Y 200.423,Z 1271.056,A -85,B 0,C 180,E1 9617.041,E2 9617.041} C_VEL
LIN {X 0,Y 201.963,Z 1268.082,A -85,B 0,C 180,E1 9610.642,E2 9610.642} C_VEL
LIN {X 0,Y 204.891,Z 1264.134,A -85,B 0,C 180,E1 9604.532,E2 9604.532} C_VEL
LIN {X 0,Y 209.43,Z 1259.184,A -85,B 0,C 180,E1 9598.657,E2 9598.657} C_VEL
LIN {X 0,Y 215.713,Z 1253.093,A -85,B 0,C 180,E1 9592.962,E2 9592.962} C_VEL
LIN {X 0,Y 224.987,Z 1244.768,A -85,B 0,C 180,E1 9586.83,E2 9586.83} C_VEL
LIN {X 0,Y 237.907,Z 1233.419,A -85,B 0,C 180,E1 9580.494,E2 9580.494} C_VEL
LIN {X 0,Y 249.644,Z 1223.098,A -85,B 0,C 180,E1 9576.018,E2 9576.018} C_VEL
LIN {X 0,Y 261.378,Z 1212.562,A -85,B 0,C 180,E1 9572.306,E2 9572.306} C_VEL
LIN {X 0,Y 274.764,Z 1200.136,A -85,B 0,C 180,E1 9568.741,E2 9568.741} C_VEL
LIN {X 0,Y 291.306,Z 1184.017,A -85,B 0,C 180,E1 9565.048,E2 9565.048} C_VEL
LIN {X 0,Y 307.329,Z 1167.112,A -85,B 0,C 180,E1 9562.022,E2 9562.022} C_VEL
LIN {X 0,Y 320.261,Z 1152.611,A -85,B 0,C 180,E1 9559.896,E2 9559.896} C_VEL
LIN {X 0,Y 333.19,Z 1137.116,A -85,B 0,C 180,E1 9557.99,E2 9557.99} C_VEL
LIN {X 0,Y 347.254,Z 1118.978,A -85,B 0,C 180,E1 9556.136,E2 9556.136} C_VEL
LIN {X 0,Y 363.537,Z 1095.756,A -85,B 0,C 180,E1 9554.222,E2 9554.222} C_VEL
LIN {X 0,Y 375.46,Z 1076.933,A -85,B 0,C 180,E1 9552.963,E2 9552.963} C_VEL
LIN {X 0,Y 386.199,Z 1058.329,A -85,B 0,C 180,E1 9551.906,E2 9551.906} C_VEL
LIN {X 0,Y 396.622,Z 1038.409,A -85,B 0,C 180,E1 9550.96,E2 9550.96} C_VEL
LIN {X 0,Y 408.081,Z 1013.825,A -85,B 0,C 180,E1 9549.996,E2 9549.996} C_VEL
